			udiTmpDWord := DINT_TO_UDINT(REAL_TO_DINT(Distance * 10000)); (*Distance*)
			Axis.PlcToDrv.MCParaWord0 := UDINT_TO_UINT(udiTmpDWord);
			Axis.PlcToDrv.MCParaWord1 := UDINT_TO_UINT(ROR(udiTmpDWord,16));

			udiTmpDWord := DINT_TO_UDINT(REAL_TO_DINT(Velocity * 1000000)); (*Maximal velocity*)
			Axis.PlcToDrv.MCParaWord2 := UDINT_TO_UINT(udiTmpDWord);
			Axis.PlcToDrv.MCParaWord3 := UDINT_TO_UINT(ROR(udiTmpDWord,16));

			udiTmpDWord := DINT_TO_UDINT(REAL_TO_DINT(Acceleration * 100000)); (*Acceleration*)
			Axis.PlcToDrv.MCParaWord4 := UDINT_TO_UINT(udiTmpDWord);
			Axis.PlcToDrv.MCParaWord5 := UDINT_TO_UINT(ROR(udiTmpDWord,16));

			udiTmpDWord := DINT_TO_UDINT(REAL_TO_DINT(Deceleration * 100000)); (*Deceleration*)
			Axis.PlcToDrv.MCParaWord6 := UDINT_TO_UINT(udiTmpDWord);
			Axis.PlcToDrv.MCParaWord7 := UDINT_TO_UINT(ROR(udiTmpDWord,16));

			udiTmpDWord := DINT_TO_UDINT(REAL_TO_DINT(Jerk * 10000)); (*Jerk*)
			Axis.PlcToDrv.MCParaWord8 := UDINT_TO_UINT(udiTmpDWord);
			Axis.PlcToDrv.MCParaWord9 := UDINT_TO_UINT(ROR(udiTmpDWord,16));
			
			LM_UptMCI(Axis);
			
			uiFbState := 2;
		ELSE
			Axis.CommandRunning := FALSE;
			uiFbState := 50; (*Error state*)
			Error := TRUE;
			ErrorID := 16#06; (*Invalid input(s)*)
		END_IF

	2:	(*Prüfen ob Befehl ausgeführt ][ Check if command has been executed*)
		IF usiOldCmdCount = usiNewCmdCount AND uiCState = 16#08 AND Axis.DrvToPlc.StateVar.6 THEN
			Done := TRUE;
			Busy := FALSE;
			Axis.PlcToDrv.MCHeader := 16#0000 + usiNewCmdCount; (*Send no operation*)
			Axis.CommandRunning := FALSE;
			uiFbState := 3;
		END_IF

	3:	IF NOT Execute THEN
			uiFbState := 0;
			Busy := FALSE;
			Done := FALSE;
		END_IF

	50:	Error := TRUE;
		Busy := FALSE;
		Done := FALSE;
		IF NOT Execute THEN
			uiFbState := 0;
			Error := FALSE;
			ErrorID := 0;
		END_IF

END_CASE

END_FUNCTION_BLOCK

// POUs/LinMot MC Function Blocks/LMmt_StartCTCommand
FUNCTION_BLOCK LMmt_StartCTCommand
VAR_INPUT
	Execute			:BOOL;	(*Execute command*)
	CTEntryID		:UINT;	(*ID of the Command Table to be started*)
END_VAR
VAR_IN_OUT
	Axis			:tstLM_Axis; (*Axis reference*)
END_VAR
VAR_OUTPUT
	Done			:BOOL;	(*Command has been executed*)
	Busy			:BOOL;	(*Command running / FB Busy*)
	Error			:BOOL;	(*Error detected*)
	ErrorID			:UINT;	(*Error ID:
							01h: Axis not ready
 							02h: Axis already has command running
 							03h: Axis has error
 							04h: Command interrupted
 							05h: Command aborted
							06h: Invalid input(s)
							*)
END_VAR
VAR
	usiOldCmdCount 	:USINT;	(*internal -> *)
	usiNewCmdCount	:USINT;	(*internal -> *)
	uiCState		:UINT;	(*internal -> *)
	uiFbState		:UINT;	(*internal -> *)
	rTrig			:LM_R_TRIG;	(*internal -> *)

 	uiCmdHeader 	:UINT := 16#2000;	(*CommandHeader (200xh) of the "Start Command Table Command (200xh)" motion command*)
END_VAR
(*Version history:
Date         	 | Version    		| Created under     	| Author          	| Remark 
------------------------------------------------------------------------------------------------------------------------------- 
2011-jul-12   	 | 1.0.0      		| V2.11.0 (Build 1016)	| fj  				| initial release
2011-sep-13   	 | 1.0.1      		| V2.11.0 (Build 1016)	| fj  				| removed check for "StandStill_LM" on Execute rising edge 
2011-dec-01   	 | 1.0.2      		| V2.11.0 (Build 1016)	| fj  				| code optimisation
2012-apr-25   	 | 1.1.0     		| V2.11.0 (Build 1016)	| fj  				| added input parameters check
*)

(*Variablen ][ variables*)
usiOldCmdCount := SHR(UINT_TO_USINT(SHL(Axis.DrvToPlc.StateVar,4)),4);
uiCState := SHR(Axis.DrvToPlc.StateVar, 8);

(*Flankenerkennung am Execute Eingang*)
(*Edge detection on Execute input*)
rTrig(CLK:=Execute);
IF rTrig.Q AND uiCState = 16#08 AND NOT Axis.CommandRunning THEN (*Start command*)
	Axis.CommandRunning := TRUE;
	Busy := TRUE;
	uiFbState := 1;
ELSIF rTrig.Q AND Busy THEN (*Restart command / New rising edge on execute input*)
	Axis.CommandRunning := TRUE;
	Busy := TRUE;
	uiFbState := 1;
ELSIF rTrig.Q AND uiCState <> 16#08 THEN (*Axis not ready*)
	uiFbState := 50; (*Error state*)
	Error := TRUE;
	ErrorID := 16#01; (*Axis not ready*)
ELSIF rTrig.Q AND Axis.CommandRunning AND NOT Busy THEN (*Axis already has a command running*)
	uiFbState := 50; (*Error state*)
	Error := TRUE;
	ErrorID := 16#02; (*Axis already has a command running*)
END_IF

IF Busy AND uiCState = 16#04 THEN
	Axis.CommandRunning := FALSE;
	uiFbState := 50;
	Error := TRUE;
	ErrorID := 16#03; (*Axis has error*)
END_IF

IF Busy AND uiCState <> 16#08 THEN
	Axis.CommandRunning := FALSE;
	uiFbState := 50; (*Error state*)
	Error := TRUE;
	ErrorID := 16#04; (*Command interupted*)
ELSIF Busy AND Axis.CommandAborted THEN
	uiFbState := 50; (*Error state*)
	Error := TRUE;
	ErrorID := 16#05; (*Command aborted*)
END_IF

(*State machine*)
CASE uiFbState OF
	0:	;

	1:	(*Check inputs on valid value*)
		IF (1 <= CTEntryID AND CTEntryID <= 255)
			THEN
			(*Befehlskopf mit CMD Count berechen und senden ][ Calculate and send command header*)
			usiNewCmdCount := (usiOldCmdCount + 1) MOD 16 ; (*MOD 16*)
			Axis.PlcToDrv.MCHeader := 16#0000; (*Reset Header*)
			Axis.PlcToDrv.MCHeader := uiCmdHeader + usiNewCmdCount;

			Axis.PlcToDrv.MCParaWord0 := CTEntryID; (*CTEntryID (line number)*)

			LM_UptMCI(Axis);

			uiFbState := 2;
		ELSE
			Axis.CommandRunning := FALSE;
			uiFbState := 50; (*Error state*)
			Error := TRUE;
			ErrorID := 16#06; (*Invalid input(s)*)
		END_IF

	2:	(*Prüfen ob Befehl ausgeführt ][ Check if command has been executed*)
		IF usiOldCmdCount = usiNewCmdCount AND uiCState = 16#08 THEN
			Done := TRUE;
			Busy := FALSE;
			Axis.PlcToDrv.MCHeader := 16#0000 + usiNewCmdCount; (*Send no operation*)
			Axis.CommandRunning := FALSE;
			uiFbState := 3;
		END_IF

	3:	IF NOT Execute THEN
			uiFbState := 0;
			Busy := FALSE;
			Done := FALSE;
		END_IF

	50:	Error := TRUE;
		Busy := FALSE;
		Done := FALSE;
		IF NOT Execute THEN
			uiFbState := 0;
			Error := FALSE;
			ErrorID := 0;
		END_IF

END_CASE

END_FUNCTION_BLOCK

// POUs/LinMot MC Function Blocks/LMmt_WriteLivePar
FUNCTION_BLOCK LMmt_WriteLivePar
VAR_INPUT
	Execute			:BOOL;	(*Execute command*)
	UPID			:UINT;	(*Parameter ID (UPID = Unique Parameter ID*)
	UPIDValue		:DINT;	(*Parameter value*)
END_VAR
VAR_IN_OUT
	Axis			:tstLM_Axis; (*Axis reference*)
END_VAR
VAR_OUTPUT
	Done			:BOOL;	(*Command has been executed*)
	Busy			:BOOL;	(*Command running / FB Busy*)
	Error			:BOOL;	(*Error detected*)
	ErrorID			:UINT;	(*Error ID:
							01h: Axis not ready
 							02h: Axis already has command running
 							03h: Axis has error
 							04h: Command interrupted
 							05h: Command aborted
							06h: Invalid input(s)
							*)
END_VAR
VAR
	usiOldCmdCount 	:USINT;	(*internal -> *)
	usiNewCmdCount	:USINT;	(*internal -> *)
	uiCState		:UINT;	(*internal -> *)
	uiFbState		:UINT;	(*internal -> *)
	rTrig			:LM_R_TRIG;	(*internal -> *)
	udiTmpDWord		:UDINT;	(*internal -> *)

 	uiCmdHeader 	:UINT := 16#0020;	(*CommandHeader (002xh) of the "Write Live Parameter (002xh)" motion command*)
END_VAR
(*Version history:
Date         	 | Version    		| Created under     	| Author          	| Remark 
------------------------------------------------------------------------------------------------------------------------------- 
2011-jul-12   	 | 1.0.0      		| V2.11.0 (Build 1016)	| fj  				| initial release 
2011-dec-01   	 | 1.0.2      		| V2.11.0 (Build 1016)	| fj  				| code optimisation
2012-apr-25   	 | 1.1.0     		| V2.11.0 (Build 1016)	| fj  				| added input parameters check
*)

(*Variablen ][ variables*)
usiOldCmdCount := SHR(UINT_TO_USINT(SHL(Axis.DrvToPlc.StateVar,4)),4);
uiCState := SHR(Axis.DrvToPlc.StateVar, 8);

(*Flankenerkennung am Execute Eingang*)
(*Edge detection on Execute input*)
rTrig(CLK:=Execute);
IF rTrig.Q AND uiCState = 16#08 AND NOT Axis.CommandRunning THEN (*Start command*)
	Axis.CommandRunning := TRUE;
	Busy := TRUE;
	uiFbState := 1;
ELSIF rTrig.Q AND Busy THEN (*Restart command / New rising edge on execute input*)
	Axis.CommandRunning := TRUE;
	Busy := TRUE;
	uiFbState := 1;
ELSIF rTrig.Q AND uiCState <> 16#08 THEN (*Axis not ready*)
	uiFbState := 50; (*Error state*)
	Error := TRUE;
	ErrorID := 16#01; (*Axis not ready*)
ELSIF rTrig.Q AND Axis.CommandRunning AND NOT Busy THEN (*Axis already has a command running*)
	uiFbState := 50; (*Error state*)
	Error := TRUE;
	ErrorID := 16#02; (*Axis already has a command running*)
END_IF

IF Busy AND uiCState = 16#04 THEN
	Axis.CommandRunning := FALSE;
	uiFbState := 50;
	Error := TRUE;
	ErrorID := 16#03; (*Axis has error*)
END_IF

IF Busy AND uiCState <> 16#08 THEN
	Axis.CommandRunning := FALSE;
	uiFbState := 50; (*Error state*)
	Error := TRUE;
	ErrorID := 16#04; (*Command interupted*)
ELSIF Busy AND Axis.CommandAborted THEN
	uiFbState := 50; (*Error state*)
	Error := TRUE;
	ErrorID := 16#05; (*Command aborted*)
END_IF

(*State machine*)
CASE uiFbState OF
	0:	;

	1:	(*Check inputs on valid value*)
		IF (0 < UPID AND UPID <= 65535)
			AND (-2147483648 <= UPIDValue AND UPIDValue <= 2147483647)
			THEN
			(*Befehlskopf mit CMD Count berechen und senden ][ Calculate and send command header*)
			usiNewCmdCount  := (usiOldCmdCount + 1) MOD 16 ; (*MOD 16*)
			Axis.PlcToDrv.MCHeader := 16#0000; (*Reset Header*)
			Axis.PlcToDrv.MCHeader := uiCmdHeader + usiNewCmdCount;

			Axis.PlcToDrv.MCParaWord0 := UPID; (*UPID number*)

			udiTmpDWord := DINT_TO_UDINT(UPIDValue); (*UPID parameter value*)
			Axis.PlcToDrv.MCParaWord1 := UDINT_TO_UINT(udiTmpDWord);
			Axis.PlcToDrv.MCParaWord2 := UDINT_TO_UINT(ROR(udiTmpDWord,16));

			LM_UptMCI(Axis);

			uiFbState := 2;
		ELSE
			Axis.CommandRunning := FALSE;
			uiFbState := 50; (*Error state*)
			Error := TRUE;
			ErrorID := 16#06; (*Invalid input(s)*)
		END_IF

	2:	(*Prüfen ob Befehl ausgeführt ][ Check if command has been executed*)
		IF usiOldCmdCount = usiNewCmdCount AND uiCState = 16#08 THEN
			Done := TRUE;
			Busy := FALSE;
			Axis.PlcToDrv.MCHeader := 16#0000 + usiNewCmdCount; (*Send no operation*)
			Axis.CommandRunning := FALSE;
			uiFbState := 3;
		END_IF

	3:	IF NOT Execute THEN
			uiFbState := 0;
			Busy := FALSE;
			Done := FALSE;
		END_IF

	50:	Error := TRUE;
		Busy := FALSE;
		Done := FALSE;
		IF NOT Execute THEN
			uiFbState := 0;
			Error := FALSE;
			ErrorID := 0;
		END_IF

END_CASE

END_FUNCTION_BLOCK

// POUs/LinMot MC Function Blocks Advanced/Unofficial_Unsupported/LMav_PVStreamLREAL
FUNCTION_BLOCK LMav_PVStreamLREAL
VAR_INPUT
	Enable 			:BOOL;	(*Enable PV streaming*)
	Position		:LREAL;	(*Setpoint position in [mm]*)
	Velocity		:LREAL;	(*Setpoint velocity in [mm/s]*)
END_VAR
VAR_IN_OUT
	Axis 			:tstLM_Axis; (*Axis*)
END_VAR
VAR_OUTPUT
	Streaming 		:BOOL;	(*Streaming / FB Busy*)
	Error 			:BOOL;	(*Error detected*)
	ErrorID			:UINT;	(*Error ID:
							01h: Axis not ready
 							02h: Axis already has command running
 							03h: Axis has error
 							04h: Command interrupted
 							05h: Command aborted
							06h: Invalid input(s)
							*)
END_VAR
VAR
	uiCState		:UINT;	(*internal -> *)
	uiFbState 		:UINT;	(*internal -> *)
	rTrig 			:LM_R_TRIG;	(*internal -> *)
	udiTmpDWord		:UDINT;	(*internal -> *)
	bTemp			:BOOL;	(*internal -> *)

	uiCmdHeader 	:UINT := 16#0310; (*internal -> CommandHeader (031xh) of the "PV Stream With Slave Generated Time Stamp (031xh)" motion command*)
END_VAR
(*Version history:
Date         	 | Version    		| Created under     	| Author          	| Remark 
------------------------------------------------------------------------------------------------------------------------------- 
2011-jul-20   	 | 1.0.0      		| V2.11.0 (Build 1016)	| fj  				| initial release
2011-sep-13   	 | 1.0.1      		| V2.11.0 (Build 1016)	| fj  				| removed check for "StandStill_LM" on Enable rising edge
2011-dec-01   	 | 1.0.2      		| V2.11.0 (Build 1016)	| fj  				| code optimisation
2012-apr-25   	 | 1.1.0     		| V2.11.0 (Build 1016)	| fj  				| removed input range check (position&velocity) / changed input data types REAL to LREAL
*)

(*Variablen ][ variables*)
uiCState := SHR(Axis.DrvToPlc.StateVar, 8);

(*Flankenerkennung am Execute Eingang*)
(*Edge detection on Execute input*)
rTrig(CLK:=Enable);
IF rTrig.Q AND uiCState = 16#08 AND NOT Axis.CommandRunning THEN (*Start command*)
	Axis.CommandRunning := TRUE;
	uiFbState := 1;
ELSIF rTrig.Q AND uiCState <> 16#08 THEN (*Axis not ready*)
	uiFbState := 50; (*Error state*)
	Error := TRUE;
	ErrorID := 16#01; (*Axis not ready*)
ELSIF rTrig.Q AND Axis.CommandRunning THEN (*Axis already has a command running*)
	uiFbState := 50; (*Error state*)
	Error := TRUE;
	ErrorID := 16#02; (*Axis already has a command running*)
END_IF

IF Streaming AND uiCState = 16#04 THEN
	Axis.CommandRunning := FALSE;
	uiFbState := 50;
	Error := TRUE;
	ErrorID := 16#03; (*Axis has error*)
END_IF

IF Streaming AND uiCState <> 16#08 THEN
	Axis.CommandRunning := FALSE;
	uiFbState := 50; (*Error state*)
	Error := TRUE;
	ErrorID := 16#04; (*Command interupted*)
ELSIF Streaming AND Axis.CommandAborted THEN
	uiFbState := 50; (*Error state*)
	Error := TRUE;
	ErrorID := 16#05; (*Command aborted*)
END_IF

(*uiState machine*)
CASE uiFbState OF
	0:	;

	1:	(*Check inputs on valid value*)
		(*Streaming*)
		bTemp := Axis.PlcToDrv.MCHeader.0;
		Axis.PlcToDrv.MCHeader := uiCmdHeader;
		Axis.PlcToDrv.MCHeader.0 := NOT bTemp;

		(*Parameter Umrechung*)
		(*Calculate parameters*)
		udiTmpDWord := DINT_TO_UDINT(LREAL_TO_DINT(Position * 10000)); (*Position*)
		Axis.PlcToDrv.MCParaWord0 := UDINT_TO_UINT(udiTmpDWord);
		Axis.PlcToDrv.MCParaWord1 := UDINT_TO_UINT(ROR(udiTmpDWord,16));

		udiTmpDWord := DINT_TO_UDINT(LREAL_TO_DINT(Velocity * 1000)); (*Velocity*)
		Axis.PlcToDrv.MCParaWord2 := UDINT_TO_UINT(udiTmpDWord);
		Axis.PlcToDrv.MCParaWord3 := UDINT_TO_UINT(ROR(udiTmpDWord,16));

		LM_UptMCI(Axis);

		Streaming := TRUE;
	
		IF NOT Enable THEN
			uiFbState := 2;
		END_IF

	2:	(*Stop streaming*)
		bTemp := Axis.PlcToDrv.MCHeader.0;
		Axis.PlcToDrv.MCHeader := 16#03F0; (*Header 03F0h (Stop Stream)*)
		Axis.PlcToDrv.MCHeader.0 := NOT bTemp;

		uiFbState := 3;

	3:	IF Axis.PlcToDrv.MCHeader.0 = Axis.DrvToPlc.StateVar.0 THEN
			Streaming := FALSE;
			Axis.PlcToDrv.MCHeader := 16#0000; (*No Operation*)
			Axis.PlcToDrv.MCHeader.0 := Axis.DrvToPlc.StateVar.0;
			Axis.CommandRunning := FALSE;
			uiFbState := 0;
		END_IF

	50:	Error := TRUE;
		Axis.PlcToDrv.MCHeader := 16#0000; (*No Operation*)
		Streaming := FALSE;
		uiFbState := 51;

	51:	 IF NOT Enable THEN
			uiFbState := 0;
			Error := FALSE;
			ErrorID := 0;
		END_IF

END_CASE

END_FUNCTION_BLOCK

// POUs/LinMot MC Function Blocks Advanced/LMav_CurrentCmdMode
FUNCTION_BLOCK LMav_CurrentCmdMode
VAR_INPUT
	Enable 			:BOOL;	(*Enable current streaming*)
	Current			:REAL;	(*Setpoint Current*)
END_VAR
VAR_IN_OUT
	Axis 			:tstLM_Axis; (*Axis reference*)
END_VAR
VAR_OUTPUT
	Streaming 		:BOOL;	(*Streaming / FB Busy*)
	Error 			:BOOL;	(*Error detected*)
	ErrorID			:UINT;	(*Error ID:
							01h: Axis not ready
 							02h: Axis already has command running
 							03h: Axis has error
 							04h: Command interrupted
 							05h: Command aborted
							06h: Invalid input(s)
							*)
END_VAR
VAR
	uiCState		:UINT;	(*internal -> *)
	uiFbState 		:UINT;	(*internal -> *)
	rTrig 			:LM_R_TRIG;	(*internal -> *)
	udiTmpDWord		:UDINT;	(*internal -> *)
	bTemp			:BOOL;	(*internal -> *)

	uiCmdHeader 	:UINT := 16#3900; (*internal -> CommandHeader (390xh) of the "Current Command Mode (390xh)" motion command*)
END_VAR
(*Version history:
Date         	 | Version    		| Created under     	| Author          	| Remark 
------------------------------------------------------------------------------------------------------------------------------- 
2011-jul-20   	 | 1.0.0      		| V2.11.0 (Build 1016)	| fj  				| initial release
2011-sep-13   	 | 1.0.1      		| V2.11.0 (Build 1016)	| fj  				| removed check for "StandStill_LM" on Execute rising edge
2011-dec-01   	 | 1.0.2      		| V2.11.0 (Build 1016)	| fj  				| code optimisation
2012-apr-25   	 | 1.1.0     		| V2.11.0 (Build 1016)	| fj  				| added input parameters check
*)

(*Variablen ][ variables*)
uiCState := SHR(Axis.DrvToPlc.StateVar, 8);

(*Flankenerkennung am Execute Eingang*)
(*Edge detection on Execute input*)
rTrig(CLK:=Enable);
IF rTrig.Q AND uiCState = 16#08 AND NOT Axis.CommandRunning THEN (*Start command*)
	Axis.CommandRunning := TRUE;
	uiFbState := 1;
ELSIF rTrig.Q AND uiCState <> 16#08 THEN (*Axis not ready*)
	uiFbState := 50; (*Error state*)
	Error := TRUE;
	ErrorID := 16#01; (*Axis not ready*)
ELSIF rTrig.Q AND Axis.CommandRunning THEN (*Axis already has a command running*)
	uiFbState := 50; (*Error state*)
	Error := TRUE;
	ErrorID := 16#02; (*Axis already has a command running*)
END_IF

IF Streaming AND uiCState = 16#04 THEN
	Axis.CommandRunning := FALSE;
	uiFbState := 50;
	Error := TRUE;
	ErrorID := 16#03; (*Axis has error*)
END_IF

IF Streaming AND uiCState <> 16#08 THEN
	Axis.CommandRunning := FALSE;
	uiFbState := 50; (*Error state*)
	Error := TRUE;
	ErrorID := 16#04; (*Command interupted*)
ELSIF Streaming AND Axis.CommandAborted THEN
	uiFbState := 50; (*Error state*)
	Error := TRUE;
	ErrorID := 16#05; (*Command aborted*)
END_IF

(*uiState machine*)
CASE uiFbState OF
	0:	;

	1:	(*Check inputs on valid value*)
		IF (-2147483.0 <= Current AND Current <= 2147483.0)
			THEN
			(*Streaming*)
			bTemp := Axis.PlcToDrv.MCHeader.0;
			Axis.PlcToDrv.MCHeader := uiCmdHeader;
			Axis.PlcToDrv.MCHeader.0 := NOT bTemp;

			(*Parameter Umrechung*)
			(*Calculate parameters*)
			udiTmpDWord := DINT_TO_UDINT(REAL_TO_DINT(Current * 1000)); (*Current*)
			Axis.PlcToDrv.MCParaWord0 := UDINT_TO_UINT(udiTmpDWord);
			Axis.PlcToDrv.MCParaWord1 := UDINT_TO_UINT(ROR(udiTmpDWord,16));

			LM_UptMCI(Axis);

			Streaming := TRUE;

			IF NOT Enable THEN
				uiFbState := 2;
			END_IF
		ELSE
			Axis.CommandRunning := FALSE;
			uiFbState := 50; (*Error state*)
			Error := TRUE;
			ErrorID := 16#06; (*Invalid input(s)*)
		END_IF

	2:	(*Stop streaming*)
		bTemp := Axis.PlcToDrv.MCHeader.0;
		Axis.PlcToDrv.MCHeader := 16#39F0; (*Header 39Fxh (Change to Position Controlled mode)*)
		Axis.PlcToDrv.MCHeader.0 := NOT bTemp;

		uiFbState := 3;

	3:	IF Axis.PlcToDrv.MCHeader.0 = Axis.DrvToPlc.StateVar.0 THEN
			Streaming := FALSE;
			Axis.CommandRunning := FALSE;
			Axis.PlcToDrv.MCHeader := 16#0000; (*No Operation*)
			Axis.PlcToDrv.MCHeader.0 := Axis.DrvToPlc.StateVar.0;
			uiFbState := 0;
		END_IF

	50:	Error := TRUE;
		Axis.PlcToDrv.MCHeader := 16#0000; (*No Operation*)
		Streaming := FALSE;
		uiFbState := 51;

	51:	 IF NOT Enable THEN
			uiFbState := 0;
			Error := FALSE;
			ErrorID := 0;
		END_IF

END_CASE

END_FUNCTION_BLOCK

// POUs/LinMot MC Function Blocks Advanced/LMav_Mod16BitCTPar
FUNCTION_BLOCK LMav_Mod16BitCTPar
VAR_INPUT
	Execute			:BOOL;	(*Execute command*)
	CTEntryID		:UINT;	(*Line number of the Command Table to be modified*)
	ParaOffset		:UINT;	(*Parameter offset (6 for the first)*)
	ParaValue		:INT;	(*Parameter value*)
END_VAR
VAR_IN_OUT
	Axis			:tstLM_Axis; (*Axis reference*)
END_VAR
VAR_OUTPUT
	Done			:BOOL;	(*Command has been executed*)
	Busy			:BOOL;	(*Command running / FB Busy*)
	Error			:BOOL;	(*Error detected*)
	ErrorID			:UINT;	(*Error ID:
							01h: Axis not ready
 							02h: Axis already has command running
 							03h: Axis has error
 							04h: Command interrupted
 							05h: Command aborted
							06h: Invalid input(s)
							*)
END_VAR
VAR
	usiOldCmdCount 	:USINT;	(*internal -> *)
	usiNewCmdCount	:USINT;	(*internal -> *)
	uiCState		:UINT;	(*internal -> *)
	uiFbState		:UINT;	(*internal -> *)
	rTrig			:LM_R_TRIG;	(*internal -> *)

 	uiCmdHeader 	:UINT := 16#2080;	(*CommandHeader (208xh) of the "Modify Command Table 16 bit Parameter in RAM (208xh)" motion command*)
END_VAR
(*Version history:
Date         	 | Version    		| Created under     	| Author          	| Remark 
------------------------------------------------------------------------------------------------------------------------------- 
2011-jul-12   	 | 1.0.0      		| V2.11.0 (Build 1016)	| fj  				| initial release 
2011-dec-01   	 | 1.0.2      		| V2.11.0 (Build 1016)	| fj  				| code optimisation
2012-apr-25   	 | 1.1.0     		| V2.11.0 (Build 1016)	| fj  				| added input parameters check
*)

(*Variablen ][ variables*)
usiOldCmdCount := SHR(UINT_TO_USINT(SHL(Axis.DrvToPlc.StateVar,4)),4);
uiCState := SHR(Axis.DrvToPlc.StateVar, 8);

(*Flankenerkennung am Execute Eingang*)
(*Edge detection on Execute input*)
rTrig(CLK:=Execute);
IF rTrig.Q AND uiCState = 16#08 AND NOT Axis.CommandRunning THEN (*Start command*)
	Axis.CommandRunning := TRUE;
	Busy := TRUE;
	uiFbState := 1;
ELSIF rTrig.Q AND Busy THEN (*Restart command / New rising edge on execute input*)
	Axis.CommandRunning := TRUE;
	Busy := TRUE;
	uiFbState := 1;
ELSIF rTrig.Q AND uiCState <> 16#08 THEN (*Axis not ready*)
	uiFbState := 50; (*Error state*)
	Error := TRUE;
	ErrorID := 16#01; (*Axis not ready*)
ELSIF rTrig.Q AND Axis.CommandRunning AND NOT Busy THEN (*Axis already has a command running*)
	uiFbState := 50; (*Error state*)
	Error := TRUE;
	ErrorID := 16#02; (*Axis already has a command running*)
END_IF

IF Busy AND uiCState = 16#04 THEN
	Axis.CommandRunning := FALSE;
	uiFbState := 50;
	Error := TRUE;
	ErrorID := 16#03; (*Axis has error*)
END_IF

IF Busy AND uiCState <> 16#08 THEN
	Axis.CommandRunning := FALSE;
	uiFbState := 50; (*Error state*)
	Error := TRUE;
	ErrorID := 16#04; (*Command interupted*)
ELSIF Busy AND Axis.CommandAborted THEN
	uiFbState := 50; (*Error state*)
	Error := TRUE;
	ErrorID := 16#05; (*Command aborted*)
END_IF

(*State machine*)
CASE uiFbState OF
	0:	;

	1:	(*Check inputs on valid value*)
		IF (0 < CTEntryID AND CTEntryID <= 255)
			AND (0 <= ParaOffset AND ParaOffset <= 20)
			AND (-32768 <= ParaValue AND ParaValue <= 32767)
			THEN
			(*Befehlskopf mit CMD Count berechen und senden ][ Calculate and send command header*)
			usiNewCmdCount := (usiOldCmdCount + 1) MOD 16; (*MOD 16*)
			Axis.PlcToDrv.MCHeader := 16#0000; (*Reset Header*)
			Axis.PlcToDrv.MCHeader := uiCmdHeader + usiNewCmdCount;

			Axis.PlcToDrv.MCParaWord0 := CTEntryID; (*CT_EntryID*)
			Axis.PlcToDrv.MCParaWord1 := ParaOffset; (*Parameter offset*)
			Axis.PlcToDrv.MCParaWord2 := INT_TO_UINT(ParaValue); (*Parameter value*)

			LM_UptMCI(Axis);

			uiFbState := 2;
		ELSE
			Axis.CommandRunning := FALSE;
			uiFbState := 50; (*Error state*)
			Error := TRUE;
			ErrorID := 16#06; (*Invalid input(s)*)
		END_IF

	2:	(*Prüfen ob Befehl ausgeführt ][ Check if command has been executed*)
		IF usiOldCmdCount = usiNewCmdCount AND uiCState = 16#08 THEN
			Done := TRUE;
			Busy := FALSE;
			Axis.PlcToDrv.MCHeader := 16#0000 + usiNewCmdCount; (*Send no operation*)
			Axis.CommandRunning := FALSE;
			uiFbState := 3;
		END_IF

	3:	IF NOT Execute THEN
			uiFbState := 0;
			Busy := FALSE;
			Done := FALSE;
		END_IF

	50:	Error := TRUE;
		Busy := FALSE;
		Done := FALSE;
		IF NOT Execute THEN
			uiFbState := 0;
			Error := FALSE;
			ErrorID := 0;
		END_IF

END_CASE

END_FUNCTION_BLOCK

// POUs/LinMot MC Function Blocks Advanced/LMav_Mod32BitCTPar
FUNCTION_BLOCK LMav_Mod32BitCTPar
VAR_INPUT
	Execute			:BOOL;	(*Execute command*)
	CTEntryID		:UINT;	(*Line number of the Command Table to be modified*)
	ParaOffset		:UINT;	(*Parameter offset (6 for the first)*)
	ParaValue		:DINT;	(*Parameter value*)
END_VAR
VAR_IN_OUT
	Axis			:tstLM_Axis; (*Axis reference*)
END_VAR
VAR_OUTPUT
	Done			:BOOL;	(*Command has been executed*)
	Busy			:BOOL;	(*Command running / FB Busy*)
	Error			:BOOL;	(*Error detected*)
	ErrorID			:UINT;	(*Error ID:
							01h: Axis not ready
 							02h: Axis already has command running
 							03h: Axis has error
 							04h: Command interrupted
 							05h: Command aborted
							06h: Invalid input(s)
							*)
END_VAR
VAR
	usiOldCmdCount 	:USINT;	(*internal -> *)
	usiNewCmdCount	:USINT;	(*internal -> *)
	uiCState		:UINT;	(*internal -> *)
	uiFbState		:UINT;	(*internal -> *)
	rTrig			:LM_R_TRIG;	(*internal -> *)
	udiTmpDWord		:UDINT;	(*internal -> *)

 	uiCmdHeader 	:UINT := 16#2090; 	(*CommandHeader (209xh) of the "Modify Command Table 32 bit Parameter in RAM (209xh)" motion command*)
END_VAR
(*Version history:
Date         	 | Version    		| Created under     	| Author          	| Remark 
------------------------------------------------------------------------------------------------------------------------------- 
2011-jul-12   	 | 1.0.0      		| V2.11.0 (Build 1016)	| fj  				| initial release 
2011-dec-01   	 | 1.0.2      		| V2.11.0 (Build 1016)	| fj  				| code optimisation
2012-apr-25   	 | 1.1.0     		| V2.11.0 (Build 1016)	| fj  				| added input parameters check
*)

(*Variablen ][ variables*)
usiOldCmdCount := SHR(UINT_TO_USINT(SHL(Axis.DrvToPlc.StateVar,4)),4);
uiCState := SHR(Axis.DrvToPlc.StateVar, 8);

(*Flankenerkennung am Execute Eingang*)
(*Edge detection on Execute input*)
rTrig(CLK:=Execute);
IF rTrig.Q AND uiCState = 16#08 AND NOT Axis.CommandRunning THEN (*Start command*)
	Axis.CommandRunning := TRUE;
	Busy := TRUE;
	uiFbState := 1;
ELSIF rTrig.Q AND Busy THEN (*Restart command / New rising edge on execute input*)
	Axis.CommandRunning := TRUE;
	Busy := TRUE;
	uiFbState := 1;
ELSIF rTrig.Q AND uiCState <> 16#08 THEN (*Axis not ready*)
	uiFbState := 50; (*Error state*)
	Error := TRUE;
	ErrorID := 16#01; (*Axis not ready*)
ELSIF rTrig.Q AND Axis.CommandRunning AND NOT Busy THEN (*Axis already has a command running*)
	uiFbState := 50; (*Error state*)
	Error := TRUE;
	ErrorID := 16#02; (*Axis already has a command running*)
END_IF

IF Busy AND uiCState = 16#04 THEN
	Axis.CommandRunning := FALSE;
	uiFbState := 50;
	Error := TRUE;
	ErrorID := 16#03; (*Axis has error*)
END_IF

IF Busy AND uiCState <> 16#08 THEN
	Axis.CommandRunning := FALSE;
	uiFbState := 50; (*Error state*)
	Error := TRUE;
	ErrorID := 16#04; (*Command interupted*)
ELSIF Busy AND Axis.CommandAborted THEN
	uiFbState := 50; (*Error state*)
	Error := TRUE;
	ErrorID := 16#05; (*Command aborted*)
END_IF

(*State machine*)
CASE uiFbState OF
	0:	;

	1:	(*Check inputs on valid value*)
		IF (0 < CTEntryID AND CTEntryID <= 255)
			AND (0 <= ParaOffset AND ParaOffset <= 20)
			AND (-2147483648 <= ParaValue AND ParaValue <= 2147483647)
			THEN
			(*Befehlskopf mit CMD Count berechen und senden ][ Calculate and send command header*)
			usiNewCmdCount := (usiOldCmdCount + 1) MOD 16 ; (*MOD 16*)
			Axis.PlcToDrv.MCHeader := 16#0000; (*Reset Header*)
			Axis.PlcToDrv.MCHeader := uiCmdHeader + usiNewCmdCount;

			Axis.PlcToDrv.MCParaWord0 := CTEntryID; (*CT_EntryID*)
			Axis.PlcToDrv.MCParaWord1 := ParaOffset; (*Parameter offset*)

			udiTmpDWord := DINT_TO_UDINT(ParaValue);(*Parameter value*)
			Axis.PlcToDrv.MCParaWord2 := UDINT_TO_UINT(udiTmpDWord);
			Axis.PlcToDrv.MCParaWord3 := UDINT_TO_UINT(ROR(udiTmpDWord,16));

			LM_UptMCI(Axis);

			uiFbState := 2;
		ELSE
			Axis.CommandRunning := FALSE;
			uiFbState := 50; (*Error state*)
			Error := TRUE;
			ErrorID := 16#06; (*Invalid input(s)*)
		END_IF

	2:	(*Prüfen ob Befehl ausgeführt ][ Check if command has been executed*)
		IF usiOldCmdCount = usiNewCmdCount AND uiCState = 16#08 THEN
			Done := TRUE;
			Busy := FALSE;
			Axis.PlcToDrv.MCHeader := 16#0000 + usiNewCmdCount; (*Send no operation*)
			Axis.CommandRunning := FALSE;
			uiFbState := 3;
		END_IF

	3:	IF NOT Execute THEN
			uiFbState := 0;
			Busy := FALSE;
			Done := FALSE;
		END_IF

	50:	Error := TRUE;
		Busy := FALSE;
		Done := FALSE;
		IF NOT Execute THEN
			uiFbState := 0;
			Error := FALSE;
			ErrorID := 0;
		END_IF

END_CASE

END_FUNCTION_BLOCK

// POUs/LinMot MC Function Blocks Advanced/LMav_MoveBestehorn
FUNCTION_BLOCK LMav_MoveBestehorn
VAR_INPUT
	Execute			:BOOL;	(*Execute command*)
	Position		:REAL;	(*Target position in [mm]*)
	Velocity		:REAL;	(*Maximal velocity in [m/s]*)
	Acceleration	:REAL;	(*Acceleration in [m/s^2]*)
	Jerk			:REAL;	(*Maximal jerk in [m/s^3]*)
END_VAR
VAR_IN_OUT
	Axis			:tstLM_Axis; (*Axis reference*)
END_VAR
VAR_OUTPUT
	Done			:BOOL;	(*Command has been executed*)
	Busy			:BOOL;	(*Command running / FB Busy*)
	Error           		:BOOL;	(*Error detected*)
	ErrorID 			:UINT;	(*Error ID:
							01h: Axis not ready
 							02h: Axis already has command running
 							03h: Axis has error
 							04h: Command interrupted
 							05h: Command aborted
							06h: Invalid input(s)
							*)
END_VAR
VAR
	usiOldCmdCount 	:USINT;	(*internal -> *)
	usiNewCmdCount	:USINT; 	(*internal -> *)
	uiCState           		:UINT;     	(*internal -> *)
	uiFbState		:UINT;	(*internal -> *)
	rTrig     	    		:LM_R_TRIG;	(*internal -> *)
	udiTmpDWord	:UDINT;	(*internal -> *)

 	uiCmdHeader 	:UINT := 16#0F00;	(*CommandHeader (0F0xh) of the "Bestehorn VAJ Go To Pos (0F0xh)" motion command*)
END_VAR
(*Version history:
Date         	 | Version    		| Created under     	| Author          	| Remark 
------------------------------------------------------------------------------------------------------------------------------- 
2011-jul-12   	 | 1.0.0      		| V2.11.0 (Build 1016)	| fj  				| initial release 
2011-sep-13   	 | 1.0.1      		| V2.11.0 (Build 1016)	| fj  				| removed check for "StandStill_LM" on Execute rising edge
2011-dec-01   	 | 1.0.2      		| V2.11.0 (Build 1016)	| fj  				| code optimisation
2012-apr-25   	 | 1.1.0     		| V2.11.0 (Build 1016)	| fj  				| added input parameters check
*)

(*Variablen ][ variables*)
usiOldCmdCount := SHR(UINT_TO_USINT(SHL(Axis.DrvToPlc.StateVar,4)),4);
uiCState := SHR(Axis.DrvToPlc.StateVar, 8);

(*Flankenerkennung am Execute Eingang*)
(*Edge detection on Execute input*)
rTrig(CLK:=Execute);
IF rTrig.Q AND uiCState = 16#08 AND NOT Axis.CommandRunning THEN (*Start command*)
	Axis.CommandRunning := TRUE;
	Busy := TRUE;
	uiFbState := 1;
ELSIF rTrig.Q AND Busy THEN (*Restart command / New rising edge on execute input*)
	Axis.CommandRunning := TRUE;
	Busy := TRUE;
	uiFbState := 1;
ELSIF rTrig.Q AND uiCState <> 16#08 THEN (*Axis not ready*)
	uiFbState := 50; (*Error state*)
	Error := TRUE;
	ErrorID := 16#01; (*Axis not ready*)
ELSIF rTrig.Q AND Axis.CommandRunning AND NOT Busy THEN (*Axis already has a command running*)
	uiFbState := 50; (*Error state*)
	Error := TRUE;
	ErrorID := 16#02; (*Axis already has a command running*)
END_IF

IF Busy AND uiCState = 16#04 THEN
	Axis.CommandRunning := FALSE;
	uiFbState := 50;
	Error := TRUE;
	ErrorID := 16#03; (*Axis has error*)
END_IF

IF Busy AND uiCState <> 16#08 THEN
	Axis.CommandRunning := FALSE;
	uiFbState := 50; (*Error state*)
	Error := TRUE;
	ErrorID := 16#04; (*Command interupted*)
ELSIF Busy AND Axis.CommandAborted THEN
	uiFbState := 50; (*Error state*)
	Error := TRUE;
	ErrorID := 16#05; (*Command aborted*)
END_IF

(*State machine*)
CASE uiFbState OF
	0:	;

	1:	(*Check inputs on valid value*)
		IF (-214748.0 <= Position AND Position <= 214748.0)
			AND (0.0 < Velocity AND Velocity <= 2147.0)
			AND (0.0 < Acceleration AND Acceleration <= 21474.0)
			AND (0.0 < Jerk AND Jerk <= 214740.0)
			THEN
			(*Befehlskopf mit CMD Count berechen und senden ][ Calculate and send command header*)
			usiNewCmdCount := (usiOldCmdCount + 1) MOD 16 ; (*MOD 16*)
			Axis.PlcToDrv.MCHeader := 16#0000; (*Reset Header*)
			Axis.PlcToDrv.MCHeader := uiCmdHeader + usiNewCmdCount ;

			udiTmpDWord := DINT_TO_UDINT(REAL_TO_DINT(Position * 10000)); (*Target position*)
			Axis.PlcToDrv.MCParaWord0 := UDINT_TO_UINT(udiTmpDWord);
			Axis.PlcToDrv.MCParaWord1 := UDINT_TO_UINT(ROR(udiTmpDWord,16));

			udiTmpDWord := DINT_TO_UDINT(REAL_TO_DINT(Velocity * 1000000)); (*Maximal velocity*)
			Axis.PlcToDrv.MCParaWord2 := UDINT_TO_UINT(udiTmpDWord);
			Axis.PlcToDrv.MCParaWord3 := UDINT_TO_UINT(ROR(udiTmpDWord,16));

			udiTmpDWord := DINT_TO_UDINT(REAL_TO_DINT(Acceleration * 100000)); (*Acceleration*)
			Axis.PlcToDrv.MCParaWord4 := UDINT_TO_UINT(udiTmpDWord);
			Axis.PlcToDrv.MCParaWord5 := UDINT_TO_UINT(ROR(udiTmpDWord,16));

			udiTmpDWord := DINT_TO_UDINT(REAL_TO_DINT(Jerk * 10000)); (*Jerk*)
			Axis.PlcToDrv.MCParaWord6 := UDINT_TO_UINT(udiTmpDWord);
			Axis.PlcToDrv.MCParaWord7 := UDINT_TO_UINT(ROR(udiTmpDWord,16));

			LM_UptMCI(Axis);

			uiFbState := 2;
		ELSE
			Axis.CommandRunning := FALSE;
			uiFbState := 50; (*Error state*)
			Error := TRUE;
			ErrorID := 16#06; (*Invalid input(s)*)
		END_IF

	2:	(*Prüfen ob Befehl ausgeführt ][ Check if command has been executed*)
		IF usiOldCmdCount = usiNewCmdCount AND uiCState = 16#08 AND Axis.DrvToPlc.StateVar.6 THEN
			Done := TRUE;
			Busy := FALSE;
			Axis.PlcToDrv.MCHeader := 16#0000 + usiNewCmdCount; (*Send no operation*)
			Axis.CommandRunning := FALSE;
			uiFbState := 3;
		END_IF

	3:	IF NOT Execute THEN
			uiFbState := 0;
			Busy := FALSE;
			Done := FALSE;
		END_IF

	50:	Error := TRUE;
		Busy := FALSE;
		Done := FALSE;
		IF NOT Execute THEN
			uiFbState := 0;
			Error := FALSE;
			ErrorID := 0;
		END_IF

END_CASE

END_FUNCTION_BLOCK

// POUs/LinMot MC Function Blocks Advanced/LMav_MoveSin
FUNCTION_BLOCK LMav_MoveSin
VAR_INPUT
	Execute			:BOOL;	(*Execute command*)
	Position		:REAL;	(*Target position in [mm]*)
	Velocity		:REAL;	(*Maximal velocity in [m/s]*)
	Acceleration	:REAL;	(*Acceleration in [m/s^2]*)
END_VAR
VAR_IN_OUT
	Axis			:tstLM_Axis; (*Axis reference*)
END_VAR
VAR_OUTPUT
	Done			:BOOL;	(*Command has been executed*)
	Busy			:BOOL;	(*Command running / FB Busy*)
	Error			:BOOL;	(*Error detected*)
	ErrorID			:UINT;	(*Error ID:
							01h: Axis not ready
 							02h: Axis already has command running
 							03h: Axis has error
 							04h: Command interrupted
 							05h: Command aborted
							06h: Invalid input(s)
							*)
END_VAR
VAR
	usiOldCmdCount 	:USINT;	(*internal -> *)
	usiNewCmdCount	:USINT;	(*internal -> *)
	uiCState		:UINT;	(*internal -> *)
	uiFbState		:UINT;	(*internal -> *)
	rTrig			:LM_R_TRIG;	(*internal -> *)
	udiTmpDWord		:UDINT;	(*internal -> *)

 	uiCmdHeader 	:UINT := 16#0E00;	(*CommandHeader (0E0xh) of the "Sin VA Go To Pos (0E0xh)" motion command*)
END_VAR
(*Version history:
Date         	 | Version    		| Created under     	| Author          	| Remark 
------------------------------------------------------------------------------------------------------------------------------- 
2011-jul-12   	 | 1.0.0      		| V2.11.0 (Build 1016)	| fj  				| initial release  
2011-sep-13   	 | 1.0.1      		| V2.11.0 (Build 1016)	| fj  				| removed check for "StandStill_LM" on Execute rising edge
2011-dec-01   	 | 1.0.2      		| V2.11.0 (Build 1016)	| fj  				| code optimisation
2012-apr-25   	 | 1.1.0     		| V2.11.0 (Build 1016)	| fj  				| added input parameters check
*)

(*Variablen ][ variables*)
usiOldCmdCount := SHR(UINT_TO_USINT(SHL(Axis.DrvToPlc.StateVar,4)),4);
uiCState := SHR(Axis.DrvToPlc.StateVar, 8);

(*Flankenerkennung am Execute Eingang*)
(*Edge detection on Execute input*)
rTrig(CLK:=Execute);
IF rTrig.Q AND uiCState = 16#08 AND NOT Axis.CommandRunning THEN (*Start command*)
	Axis.CommandRunning := TRUE;
	Busy := TRUE;
	uiFbState := 1;
ELSIF rTrig.Q AND Busy THEN (*Restart command / New rising edge on execute input*)
	Axis.CommandRunning := TRUE;
	Busy := TRUE;
	uiFbState := 1;
ELSIF rTrig.Q AND uiCState <> 16#08 THEN (*Axis not ready*)
	uiFbState := 50; (*Error state*)
	Error := TRUE;
	ErrorID := 16#01; (*Axis not ready*)
ELSIF rTrig.Q AND Axis.CommandRunning AND NOT Busy THEN (*Axis already has a command running*)
	uiFbState := 50; (*Error state*)
	Error := TRUE;
	ErrorID := 16#02; (*Axis already has a command running*)
END_IF

IF Busy AND uiCState = 16#04 THEN
	Axis.CommandRunning := FALSE;
	uiFbState := 50;
	Error := TRUE;
	ErrorID := 16#03; (*Axis has error*)
END_IF

IF Busy AND uiCState <> 16#08 THEN
	Axis.CommandRunning := FALSE;
	uiFbState := 50; (*Error state*)
	Error := TRUE;
	ErrorID := 16#04; (*Command interupted*)
ELSIF Busy AND Axis.CommandAborted THEN
	uiFbState := 50; (*Error state*)
	Error := TRUE;
	ErrorID := 16#05; (*Command aborted*)
END_IF

(*State machine*)
CASE uiFbState OF
0:	;

1:	(*Check inputs on valid value*)
	IF (-214748.0 <= Position AND Position <= 214748.0)
		AND (0.0 < Velocity AND Velocity <= 2147.0)
		AND (0.0 < Acceleration AND Acceleration <= 21474.0)
		THEN
		(*Befehlskopf mit CMD Count berechen und senden ][ Calculate and send command header*)
		usiNewCmdCount := (usiOldCmdCount + 1) MOD 16 ; (*MOD 16*)
		Axis.PlcToDrv.MCHeader := 16#0000; (*Reset Header*)
		Axis.PlcToDrv.MCHeader := uiCmdHeader + usiNewCmdCount;

		udiTmpDWord := DINT_TO_UDINT(REAL_TO_DINT(Position * 10000)); (*Target position*)
		Axis.PlcToDrv.MCParaWord0 := UDINT_TO_UINT(udiTmpDWord);
		Axis.PlcToDrv.MCParaWord1:= UDINT_TO_UINT(ROR(udiTmpDWord,16));

		udiTmpDWord := DINT_TO_UDINT(REAL_TO_DINT(Velocity * 1000000)); (*Maximal velocity*)
		Axis.PlcToDrv.MCParaWord2 := UDINT_TO_UINT(udiTmpDWord);
		Axis.PlcToDrv.MCParaWord3 := UDINT_TO_UINT(ROR(udiTmpDWord,16));

		udiTmpDWord := DINT_TO_UDINT(REAL_TO_DINT(Acceleration * 100000)); (*Acceleration*)
		Axis.PlcToDrv.MCParaWord4 := UDINT_TO_UINT(udiTmpDWord);
		Axis.PlcToDrv.MCParaWord5 := UDINT_TO_UINT(ROR(udiTmpDWord,16));

		LM_UptMCI(Axis);

		uiFbState := 2;
	ELSE
		Axis.CommandRunning := FALSE;
		uiFbState := 50; (*Error state*)
		Error := TRUE;
		ErrorID := 16#06; (*Invalid input(s)*)
	END_IF

2:	(*Prüfen ob Befehl ausgeführt ][ Check if command has been executed*)
	IF usiOldCmdCount = usiNewCmdCount AND uiCState = 16#08 AND Axis.DrvToPlc.StateVar.6 THEN
		Done := TRUE;
		Busy := FALSE;
		Axis.PlcToDrv.MCHeader := 16#0000 + usiNewCmdCount; (*Send no operation*)
		Axis.CommandRunning := FALSE;
		uiFbState := 3;
	END_IF

3:	IF NOT Execute THEN
		uiFbState := 0;
		Busy := FALSE;
		Done := FALSE;
	END_IF

50:	Error := TRUE;
	Busy := FALSE;
	Done := FALSE;
	IF NOT Execute THEN
		uiFbState := 0;
		Error := FALSE;
		ErrorID := 0;
	END_IF

END_CASE

END_FUNCTION_BLOCK

// POUs/LinMot MC Function Blocks Advanced/LMav_PStream
FUNCTION_BLOCK LMav_PStream
VAR_INPUT
	Enable 			:BOOL;	(*Enable P streaming*)
	Position		:REAL;	(*Setpoint Position in [mm]*)
END_VAR
VAR_IN_OUT
	Axis 			:tstLM_Axis; (*Axis*)
END_VAR
VAR_OUTPUT
	Streaming 		:BOOL;	(*Streaming / FB Busy*)
	Error 			:BOOL;	(*Error detected*)
	ErrorID			:UINT;	(*Error ID:
							01h: Axis not ready
 							02h: Axis already has command running
 							03h: Axis has error
 							04h: Command interrupted
 							05h: Command aborted
							06h: Invalid input(s)
							*)
END_VAR
VAR
	uiCState		:UINT;	(*internal -> *)
	uiFbState 		:UINT;	(*internal -> *)
	rTrig 			:LM_R_TRIG;	(*internal -> *)
	udiTmpDWord		:UDINT;	(*internal -> *)
	bTemp			:BOOL;	(*internal -> *)

	uiCmdHeader 	:UINT := 16#0300; (*internal -> CommandHeader (030xh) of the "P Stream With Slave Generated Time Stamp (030xh)" motion command*)
END_VAR
(*Version history:
Date         	 | Version    		| Created under     	| Author          	| Remark 
------------------------------------------------------------------------------------------------------------------------------- 
2011-jul-20   	 | 1.0.0      		| V2.11.0 (Build 1016)	| fj  				| initial release
2011-sep-13   	 | 1.0.1      		| V2.11.0 (Build 1016)	| fj  				| removed check for "StandStill_LM" on Enable rising edge
2011-dec-01   	 | 1.0.2      		| V2.11.0 (Build 1016)	| fj  				| code optimisation
2012-apr-25   	 | 1.1.0     		| V2.11.0 (Build 1016)	| fj  				| added input parameters check
*)

(*Variablen ][ variables*)
uiCState := SHR(Axis.DrvToPlc.StateVar, 8);

(*Flankenerkennung am Execute Eingang*)
(*Edge detection on Execute input*)
rTrig(CLK:=Enable);
IF rTrig.Q AND uiCState = 16#08 AND NOT Axis.CommandRunning THEN (*Start command*)
	Axis.CommandRunning := TRUE;
	uiFbState := 1;
ELSIF rTrig.Q AND uiCState <> 16#08 THEN (*Axis not ready*)
	uiFbState := 50; (*Error state*)
	Error := TRUE;
	ErrorID := 16#01; (*Axis not ready*)
ELSIF rTrig.Q AND Axis.CommandRunning THEN (*Axis already has a command running*)
	uiFbState := 50; (*Error state*)
	Error := TRUE;
	ErrorID := 16#02; (*Axis already has a command running*)
END_IF

IF Streaming AND uiCState = 16#04 THEN
	Axis.CommandRunning := FALSE;
	uiFbState := 50;
	Error := TRUE;
	ErrorID := 16#03; (*Axis has error*)
END_IF

IF Streaming AND uiCState <> 16#08 THEN
	Axis.CommandRunning := FALSE;
	uiFbState := 50; (*Error state*)
	Error := TRUE;
	ErrorID := 16#04; (*Command interupted*)
ELSIF Streaming AND Axis.CommandAborted THEN
	uiFbState := 50; (*Error state*)
	Error := TRUE;
	ErrorID := 16#05; (*Command aborted*)
END_IF

(*uiState machine*)
CASE uiFbState OF
	0:	;

	1:	(*Check inputs on valid value*)
		IF (-214748.0 <= Position AND Position <= 214748.0)
			THEN
			(*Streaming*)
			bTemp := Axis.PlcToDrv.MCHeader.0;
			Axis.PlcToDrv.MCHeader := uiCmdHeader;
			Axis.PlcToDrv.MCHeader.0 := NOT bTemp;

			(*Parameter Umrechung*)
			(*Calculate parameters*)
			udiTmpDWord := DINT_TO_UDINT(REAL_TO_DINT(Position * 10000)); (*Position*)
			Axis.PlcToDrv.MCParaWord0 := UDINT_TO_UINT(udiTmpDWord);
			Axis.PlcToDrv.MCParaWord1 := UDINT_TO_UINT(ROR(udiTmpDWord,16));

			LM_UptMCI(Axis);

			Streaming := TRUE;
		
			IF NOT Enable THEN
				uiFbState := 2;
			END_IF
		ELSE
			Axis.CommandRunning := FALSE;
			uiFbState := 50; (*Error state*)
			Error := TRUE;
			ErrorID := 16#06; (*Invalid input(s)*)
		END_IF

	2:	(*Stop streaming*)
		bTemp := Axis.PlcToDrv.MCHeader.0;
		Axis.PlcToDrv.MCHeader := 16#03F0; (*Header 03F0h (Stop Stream)*)
		Axis.PlcToDrv.MCHeader.0 := NOT bTemp;

		uiFbState := 3;

	3:	IF Axis.PlcToDrv.MCHeader.0 = Axis.DrvToPlc.StateVar.0 THEN
			Streaming := FALSE;
			Axis.PlcToDrv.MCHeader := 16#0000; (*No Operation*)
			Axis.PlcToDrv.MCHeader.0 := Axis.DrvToPlc.StateVar.0;
			Axis.CommandRunning := FALSE;
			uiFbState := 0;
		END_IF

	50:	Error := TRUE;
		Axis.PlcToDrv.MCHeader := 16#0000; (*No Operation*)
		Streaming := FALSE;
		uiFbState := 51;

	51:	 IF NOT Enable THEN
			uiFbState := 0;
			Error := FALSE;
			ErrorID := 0;
		END_IF

END_CASE

END_FUNCTION_BLOCK

// POUs/LinMot MC Function Blocks Advanced/LMav_PVStream
FUNCTION_BLOCK LMav_PVStream
VAR_INPUT
	Enable 			:BOOL;	(*Enable PV streaming*)
	Position		:REAL;	(*Setpoint position in [mm]*)
	Velocity		:REAL;	(*Setpoint velocity in [mm/s]*)
END_VAR
VAR_IN_OUT
	Axis 			:tstLM_Axis; (*Axis*)
END_VAR
VAR_OUTPUT
	Streaming 		:BOOL;	(*Streaming / FB Busy*)
	Error 			:BOOL;	(*Error detected*)
	ErrorID			:UINT;	(*Error ID:
							01h: Axis not ready
 							02h: Axis already has command running
 							03h: Axis has error
 							04h: Command interrupted
 							05h: Command aborted
							06h: Invalid input(s)
							*)
END_VAR
VAR
	uiCState		:UINT;	(*internal -> *)
	uiFbState 		:UINT;	(*internal -> *)
	rTrig 			:LM_R_TRIG;	(*internal -> *)
	udiTmpDWord		:UDINT;	(*internal -> *)
	bTemp			:BOOL;	(*internal -> *)

	uiCmdHeader 	:UINT := 16#0310; (*internal -> CommandHeader (031xh) of the "PV Stream With Slave Generated Time Stamp (031xh)" motion command*)
END_VAR
(*Version history:
Date         	 | Version    		| Created under     	| Author          	| Remark 
------------------------------------------------------------------------------------------------------------------------------- 
2011-jul-20   	 | 1.0.0      		| V2.11.0 (Build 1016)	| fj  				| initial release
2011-sep-13   	 | 1.0.1      		| V2.11.0 (Build 1016)	| fj  				| removed check for "StandStill_LM" on Enable rising edge
2011-dec-01   	 | 1.0.2      		| V2.11.0 (Build 1016)	| fj  				| code optimisation
2012-apr-25   	 | 1.1.0     		| V2.11.0 (Build 1016)	| fj  				| added input parameters check
*)

(*Variablen ][ variables*)
uiCState := SHR(Axis.DrvToPlc.StateVar, 8);

(*Flankenerkennung am Execute Eingang*)
(*Edge detection on Execute input*)
rTrig(CLK:=Enable);
IF rTrig.Q AND uiCState = 16#08 AND NOT Axis.CommandRunning THEN (*Start command*)
	Axis.CommandRunning := TRUE;
	uiFbState := 1;
ELSIF rTrig.Q AND uiCState <> 16#08 THEN (*Axis not ready*)
	uiFbState := 50; (*Error state*)
	Error := TRUE;
	ErrorID := 16#01; (*Axis not ready*)
ELSIF rTrig.Q AND Axis.CommandRunning THEN (*Axis already has a command running*)
	uiFbState := 50; (*Error state*)
	Error := TRUE;
	ErrorID := 16#02; (*Axis already has a command running*)
END_IF

IF Streaming AND uiCState = 16#04 THEN
	Axis.CommandRunning := FALSE;
	uiFbState := 50;
	Error := TRUE;
	ErrorID := 16#03; (*Axis has error*)
END_IF

IF Streaming AND uiCState <> 16#08 THEN
	Axis.CommandRunning := FALSE;
	uiFbState := 50; (*Error state*)
	Error := TRUE;
	ErrorID := 16#04; (*Command interupted*)
ELSIF Streaming AND Axis.CommandAborted THEN
	uiFbState := 50; (*Error state*)
	Error := TRUE;
	ErrorID := 16#05; (*Command aborted*)
END_IF

(*uiState machine*)
CASE uiFbState OF
	0:	;

	1:	(*Check inputs on valid value*)
		IF (-214748.0 <= Position AND Position <= 214748.0)
			AND (-2147.0 <= Velocity AND Velocity <= 2147.0)
			THEN
			(*Streaming*)
			bTemp := Axis.PlcToDrv.MCHeader.0;
			Axis.PlcToDrv.MCHeader := uiCmdHeader;
			Axis.PlcToDrv.MCHeader.0 := NOT bTemp;

			(*Parameter Umrechung*)
			(*Calculate parameters*)
			udiTmpDWord := DINT_TO_UDINT(REAL_TO_DINT(Position * 10000)); (*Position*)
			Axis.PlcToDrv.MCParaWord0 := UDINT_TO_UINT(udiTmpDWord);
			Axis.PlcToDrv.MCParaWord1 := UDINT_TO_UINT(ROR(udiTmpDWord,16));

			udiTmpDWord := DINT_TO_UDINT(REAL_TO_DINT(Velocity * 1000)); (*Velocity*)
			Axis.PlcToDrv.MCParaWord2 := UDINT_TO_UINT(udiTmpDWord);
			Axis.PlcToDrv.MCParaWord3 := UDINT_TO_UINT(ROR(udiTmpDWord,16));

			LM_UptMCI(Axis);

			Streaming := TRUE;
		
			IF NOT Enable THEN
				uiFbState := 2;
			END_IF
		ELSE
			Axis.CommandRunning := FALSE;
			uiFbState := 50; (*Error state*)
			Error := TRUE;
			ErrorID := 16#06; (*Invalid input(s)*)
		END_IF

	2:	(*Stop streaming*)
		bTemp := Axis.PlcToDrv.MCHeader.0;
		Axis.PlcToDrv.MCHeader := 16#03F0; (*Header 03F0h (Stop Stream)*)
		Axis.PlcToDrv.MCHeader.0 := NOT bTemp;

		uiFbState := 3;

	3:	IF Axis.PlcToDrv.MCHeader.0 = Axis.DrvToPlc.StateVar.0 THEN
			Streaming := FALSE;
			Axis.PlcToDrv.MCHeader := 16#0000; (*No Operation*)
			Axis.PlcToDrv.MCHeader.0 := Axis.DrvToPlc.StateVar.0;
			Axis.CommandRunning := FALSE;
			uiFbState := 0;
		END_IF

	50:	Error := TRUE;
		Axis.PlcToDrv.MCHeader := 16#0000; (*No Operation*)
		Streaming := FALSE;
		uiFbState := 51;

	51:	 IF NOT Enable THEN
			uiFbState := 0;
			Error := FALSE;
			ErrorID := 0;
		END_IF

END_CASE

END_FUNCTION_BLOCK

// POUs/LinMot MC Function Blocks Advanced/LMav_RunCurve
FUNCTION_BLOCK LMav_RunCurve
VAR_INPUT
	Execute			:BOOL;	(*Execute command)*)
	CurveID			:UINT;	(*Curve ID*)
	CurveOffset		:REAL;	(*Offset in [mm]*)
	TimeScale		:REAL;	(*Time scale (0-200%)*)
	AmplitudeScale	:REAL;	(*Amplitude scale (-2000% to +2000%*)
END_VAR
VAR_IN_OUT
	Axis 			:tstLM_Axis; (*Axis*)
END_VAR
VAR_OUTPUT
	Done			:BOOL;	(*Command has been executed*)
	Busy			:BOOL;	(*Command running / FB Busy*)
	Error			:BOOL;	(*Error detected*)
	ErrorID			:UINT;	(*Error ID:
							01h: Axis not ready
 							02h: Axis already has command running
 							03h: Axis has error
 							04h: Command interrupted
 							05h: Command aborted
							06h: Invalid input(s)
							*)
END_VAR
VAR
	usiOldCmdCount 	:USINT;	(*internal -> *)
	usiNewCmdCount	:USINT;	(*internal -> *)
	uiCState		:UINT;	(*internal -> *)
	uiFbState		:UINT;	(*internal -> *)
	rTrig			:LM_R_TRIG;	(*internal -> *)
	udiTmpDWord		:UDINT;	(*internal -> *)

 	uiCmdHeader 	:UINT := 16#0440;	(*CommandHeader (044xh) of the "Time Curve With Adjustable Offset, Time Scale & Amplitude Scale (044xh)" motion command*)
END_VAR
(*Version history:
Date         	 | Version    		| Created under     	| Author          	| Remark 
------------------------------------------------------------------------------------------------------------------------------- 
2011-jul-12   	 | 1.0.0      		| V2.11.0 (Build 1016)	| fj  				| initial release
2011-sep-13   	 | 1.0.1      		| V2.11.0 (Build 1016)	| fj  				| removed check for "StandStill_LM" on Execute rising edge
2011-dec-01   	 | 1.0.2      		| V2.11.0 (Build 1016)	| fj  				| code optimisation
2012-apr-25   	 | 1.1.0     		| V2.11.0 (Build 1016)	| fj  				| added input parameters check
*)

(*Variablen ][ variables*)
usiOldCmdCount := SHR(UINT_TO_USINT(SHL(Axis.DrvToPlc.StateVar,4)),4);
uiCState := SHR(Axis.DrvToPlc.StateVar, 8);

(*Flankenerkennung am Execute Eingang*)
(*Edge detection on Execute input*)
rTrig(CLK:=Execute);
IF rTrig.Q AND uiCState = 16#08 AND NOT Axis.CommandRunning THEN (*Start command*)
	Axis.CommandRunning := TRUE;
	Busy := TRUE;
	uiFbState := 1;
ELSIF rTrig.Q AND Busy THEN (*Restart command / New rising edge on execute input*)
	Axis.CommandRunning := TRUE;
	Busy := TRUE;
	uiFbState := 1;
ELSIF rTrig.Q AND uiCState <> 16#08 THEN (*Axis not ready*)
	uiFbState := 50; (*Error state*)
	Error := TRUE;
	ErrorID := 16#01; (*Axis not ready*)
ELSIF rTrig.Q AND Axis.CommandRunning AND NOT Busy THEN (*Axis already has a command running*)
	uiFbState := 50; (*Error state*)
	Error := TRUE;
	ErrorID := 16#02; (*Axis already has a command running*)
END_IF

IF Busy AND uiCState = 16#04 THEN
	Axis.CommandRunning := FALSE;
	uiFbState := 50;
	Error := TRUE;
	ErrorID := 16#03; (*Axis has error*)
END_IF

IF Busy AND uiCState <> 16#08 THEN
	Axis.CommandRunning := FALSE;
	uiFbState := 50; (*Error state*)
	Error := TRUE;
	ErrorID := 16#04; (*Command interupted*)
ELSIF Busy AND Axis.CommandAborted THEN
	uiFbState := 50; (*Error state*)
	Error := TRUE;
	ErrorID := 16#05; (*Command aborted*)
END_IF

(*State machine*)
CASE uiFbState OF
	0:	;

	1:	(*Check inputs on valid value*)
		IF (1 <= CurveID AND CurveID <= 255)
			AND (-214748.0 <= CurveOffset AND CurveOffset <= 214748.0)
			AND (0.0 < TimeScale AND TimeScale <= 200.0)
			AND (-2000.0 <= AmplitudeScale AND AmplitudeScale <= 2000.0)
			THEN
			(*Befehlskopf mit CMD Count berechen und senden ][ Calculate and send command header*)
			usiNewCmdCount := (usiOldCmdCount + 1) MOD 16 ; (*MOD 16*)
			Axis.PlcToDrv.MCHeader := 16#0000; (*Reset Header*)
			Axis.PlcToDrv.MCHeader := uiCmdHeader + usiNewCmdCount;

			Axis.PlcToDrv.MCParaWord0 := CurveID; (*CurveID*)

			udiTmpDWord := DINT_TO_UDINT(REAL_TO_DINT(CurveOffset * 10000)); (*Curve Offset*)
			Axis.PlcToDrv.MCParaWord1 := UDINT_TO_UINT(udiTmpDWord);
			Axis.PlcToDrv.MCParaWord2 := UDINT_TO_UINT(ROR(udiTmpDWord,16));

			Axis.PlcToDrv.MCParaWord3 := REAL_TO_UINT(TimeScale * 100); (*Time Scale*)
			Axis.PlcToDrv.MCParaWord4 := REAL_TO_UINT(AmplitudeScale * 10); (*Amplitude Scale*)

			LM_UptMCI(Axis);

			uiFbState := 2;
		ELSE
			Axis.CommandRunning := FALSE;
			uiFbState := 50; (*Error state*)
			Error := TRUE;
			ErrorID := 16#06; (*Invalid input(s)*)
		END_IF

	2:	(*Prüfen ob Befehl ausgeführt ][ Check if command has been executed*)
		IF usiOldCmdCount = usiNewCmdCount AND uiCState = 16#08 AND Axis.DrvToPlc.StateVar.6 THEN
			Done := TRUE;
			Busy := FALSE;
			Axis.PlcToDrv.MCHeader := 16#0000 + usiNewCmdCount; (*Send no operation*)
			Axis.CommandRunning := FALSE;
			uiFbState := 3;
		END_IF

	3:	IF NOT Execute THEN
			uiFbState := 0;
			Busy := FALSE;
			Done := FALSE;
		END_IF

	50:	Error := TRUE;
		Busy := FALSE;
		Done := FALSE;
		IF NOT Execute THEN
			uiFbState := 0;
			Error := FALSE;
			ErrorID := 0;
		END_IF

END_CASE

END_FUNCTION_BLOCK

// POUs/Rotary Motors/LMct_RotaryMotorControl
FUNCTION_BLOCK LMct_RotaryMotorControl
VAR_INPUT
	SwitchOn		    :BOOL;	(*Switch on motor*)
	Home				:BOOL;	(*Start homing procedure*)
	ErrorAcknowledge	:BOOL;	(*Error acknowledge*)
	JogPlus				:BOOL;	(*Jog move postive*)
	JogMinus			:BOOL;	(*Jog move negative*)
	SetReference		:BOOL;	(*Set rotary motor reference*)
	ReferenceAngle		:DINT;	(*[Units]*)
	ModuloFactor		:DINT;	(*[Units]*)
END_VAR
VAR_IN_OUT
	Axis	       		:tstLM_Axis; (*Axis reference*)
END_VAR
VAR_OUTPUT
	OperationEnabled	:BOOL;	(*Axis powered on*)
	SwitchOnLocked		:BOOL;	(*Switch on locked*)
	Homed     	      	:BOOL;	(*Axis has reference*)
	ReferenceSet		:BOOL;	(*Reference Set*)
	MotionActive		:BOOL;	(*Motion active (Setpoint generation (VAI, curve) active)*)
	Jogging				:BOOL;	(*Axis is moving in jog mode*)
	Warning         	:BOOL;	(*Warning detected*)
	Error          		:BOOL;	(*Error detected*)
	ErrorCode      		:UINT;	(*Error code, see MotionCtrlSW manual*)
	MotorDemandAngle  	:DINT;	(*Demand angle in [Units]*)
	MotorActualAngle  	:DINT;	(*Actual position in [Units]*)
	NrOfRevolutions		:DINT;	(*Number of revolutions*)
	ActualCurrent   	:REAL;	(*Actual motor current in [A]*)
END_VAR
VAR
	uiState        		:UINT;	(*internal -> Current state of the drive*)
	rTrigHome 			:LM_R_TRIG;	(*internal ->*)
	fTrigHome 			:LM_F_TRIG;	(*internal ->*)
	rTrigSetReference	:LM_R_TRIG;	(*internal ->*)
	dOldMotorDemandAngle:DINT;	(*internal ->*)
END_VAR
(*Version history:
Date         	 | Version    		| Created under     	| Author          	| Remark 
------------------------------------------------------------------------------------------------------------------------------- 
2014-oct-20   	 | 1.0.0.0     		| v3.1.4014.0			| fj  				| initial version
2015-feb-04   	 | 1.0.0.1     		| v3.1.4014.0			| fj  				| avoid demand angle == modulo factor -> set demand angle to 0
*)

(*Eingänge zuweisen/lesen ][ Read and allocate inputs*)
	(*Calculate motor demand angle and number of revolutions*)
	MotorDemandAngle := MotorDemandAngle + (Axis.DrvToPlc.ComDemandPosition - dOldMotorDemandAngle);
	dOldMotorDemandAngle := Axis.DrvToPlc.ComDemandPosition;
	IF MotorDemandAngle < 0 THEN
		MotorDemandAngle := MotorDemandAngle + ModuloFactor;
		IF NrOfRevolutions = -2147483648 THEN //Prevent DINT underflow
			NrOfRevolutions := 2147483647;
		ELSE
			NrOfRevolutions := NrOfRevolutions - 1;
		END_IF;
	ELSIF MotorDemandAngle > ModuloFactor THEN
		MotorDemandAngle := MotorDemandAngle - ModuloFactor;
		IF NrOfRevolutions = 2147483647 THEN //Prevent DINT overflow
			NrOfRevolutions := -2147483648;
		ELSE
			NrOfRevolutions := NrOfRevolutions + 1;
		END_IF;
	ELSIF MotorDemandAngle = ModuloFactor THEN  (*If the demand angle is exactly the modulo factor set demand angle to 0*)
		MotorDemandAngle :=0;
		IF NrOfRevolutions = 2147483647 THEN (*Prevent DINT overflow*)
			NrOfRevolutions := -2147483648;
		ELSE
			NrOfRevolutions := NrOfRevolutions + 1;
		END_IF;
	END_IF;

	(*Calculate motor actual angle*)
	MotorActualAngle := MotorDemandAngle - (Axis.DrvToPlc.ComDemandPosition - Axis.DrvToPlc.ComActualPosition);
	IF MotorActualAngle < 0 THEN
		MotorActualAngle := MotorActualAngle + ModuloFactor;
	ELSIF MotorActualAngle > ModuloFactor THEN
		MotorActualAngle := MotorActualAngle - ModuloFactor;
	END_IF;

	(*Workaround for different XML current definitions (16Bit/32Bit)*)
	IF Axis.DrvToPlc.ComActualCurrent32 = 0 AND Axis.DrvToPlc.ComActualCurrent16 = 0 THEN
		ActualCurrent := 0;
	ELSIF Axis.DrvToPlc.ComActualCurrent32 <> 0 AND Axis.DrvToPlc.ComActualCurrent16 = 0 THEN
		ActualCurrent := DINT_TO_REAL(Axis.DrvToPlc.ComActualCurrent32)/1000;
	ELSIF Axis.DrvToPlc.ComActualCurrent32 = 0 AND Axis.DrvToPlc.ComActualCurrent16 <> 0 THEN
		ActualCurrent := INT_TO_REAL(Axis.DrvToPlc.ComActualCurrent16)/1000;
	ELSE
		ActualCurrent := DINT_TO_REAL(Axis.DrvToPlc.ComActualCurrent32)/1000; (*If both 16/32Bit currents aren't 0 32Bit has higher priority*)
	END_IF

(*Variablen ][ variables*)
	uiState := SHR(Axis.DrvToPlc.StateVar, 8);
	SwitchOnLocked := Axis.DrvToPlc.StatusWord.6;
	Warning := Axis.DrvToPlc.StatusWord.7;
	MotionActive := Axis.DrvToPlc.StatusWord.13;
	OperationEnabled := Axis.DrvToPlc.StatusWord.0;

(*=============================================================================
*  State Machine
===============================================================================*)    

CASE uiState OF
	(*Not Ready to Switch On*)
	00:	Axis.AxisState := Disabled_LM;

	(*State 4: Error*)
	04:	ErrorCode := UINT_TO_USINT(Axis.DrvToPlc.StateVar);
		Error := TRUE;
		Axis.AxisState := ErrorStop_LM;

	(*State 8: Operation Enabled*)
	08:	Homed := Axis.DrvToPlc.StateVar.7;
		IF Axis.DrvToPlc.StatusWord.13 AND NOT (Axis.AxisState = Stopping_LM) THEN
			Axis.AxisState := DiscreteMotion_LM;
		ELSIF NOT Axis.DrvToPlc.StatusWord.13 AND NOT (Axis.AxisState = Stopping_LM) THEN
			Axis.AxisState := StandStill_LM;
		END_IF

	(*State 9: Homing*)
	09:	Axis.AxisState := Homing_LM;
		IF Axis.DrvToPlc.StateVar = 16#090F THEN
            ReferenceSet := TRUE;
            IF ModuloFactor > 0 THEN (*prevent division by 0*)
                NrOfRevolutions := (ReferenceAngle - (ReferenceAngle MOD ModuloFactor)) / ModuloFactor;
            END_IF;
            MotorDemandAngle := ReferenceAngle MOD ModuloFactor;
            MotorActualAngle := MotorDemandAngle - (Axis.DrvToPlc.ComDemandPosition - Axis.DrvToPlc.ComActualPosition); (*Act angle = demand angle - position error*)
            IF MotorActualAngle < 0 THEN
                MotorActualAngle := MotorActualAngle + ModuloFactor;
            ELSIF MotorActualAngle > ModuloFactor THEN
                MotorActualAngle := MotorActualAngle - ModuloFactor;
            END_IF;
            Axis.PlcToDrv.ControlWord.11 := FALSE;
        END_IF;

	(*State 14: Error Behaviour QuickStop*)
	14:	Axis.AxisState := ErrorStop_LM;

	(*State 16: Jogging +*)
	16:	Axis.AxisState := Jogging_LM;

	(*State 17: Jogging -*)
	17:	Axis.AxisState := Jogging_LM;

END_CASE;


(*Wenn der drive nicht im Fehlerzustand ist, werden Error und ErrorCode auf Null gesetzt*)
(*If the drive is not in Error state, Error and ErrorCode are set to zero*)
IF uiState <> 16#04 THEN
	Error := FALSE;
	ErrorCode := 16#00;
END_IF;

IF uiState <> 16#08 THEN
	Axis.PlcToDrv.MCHeader := 16#0000; (*Reset Header to prevent "MC Cmd in wrong state" error*)
	Axis.CommandRunning := FALSE;
	Axis.CommandAborted := FALSE;
END_IF;

(*Switch On*)
Axis.PlcToDrv.ControlWord.0 := SwitchOn;
IF NOT Axis.PlcToDrv.ControlWord.0 AND NOT (uiState = 4 OR uiState = 14) THEN
	Axis.AxisState := Disabled_LM;
END_IF

(*Set Reference*)
rTrigSetReference(CLK:=SetReference);
IF rTrigSetReference.Q THEN
    ReferenceSet := TRUE;
    IF ModuloFactor > 0 THEN (*prevent division by 0*)
        NrOfRevolutions := (ReferenceAngle - (ReferenceAngle MOD ModuloFactor)) / ModuloFactor;
    END_IF;
    
    MotorDemandAngle := ReferenceAngle MOD ModuloFactor;
    IF MotorDemandAngle < 0 THEN
        MotorDemandAngle := MotorDemandAngle + ModuloFactor;
    ELSIF MotorDemandAngle > ModuloFactor THEN
        MotorDemandAngle := MotorDemandAngle - ModuloFactor;
    END_IF;

    MotorActualAngle := MotorDemandAngle - (Axis.DrvToPlc.ComDemandPosition - Axis.DrvToPlc.ComActualPosition); (*Istwinkel = Sollwinkel - Schleppfehler*)
    IF MotorActualAngle < 0 THEN
        MotorActualAngle := MotorActualAngle + ModuloFactor;
    ELSIF MotorActualAngle > ModuloFactor THEN
        MotorActualAngle := MotorActualAngle - ModuloFactor;
    END_IF;
END_IF;

(*Home*)
rTrigHome(CLK:=Home);
fTrigHome(CLK:=Home);
IF rTrigHome.Q THEN
	Axis.PlcToDrv.ControlWord.11 := TRUE;
END_IF
IF fTrigHome.Q  THEN
	Axis.PlcToDrv.ControlWord.11 := FALSE;
END_IF

IF uiState = 16#09 OR (Axis.PlcToDrv.ControlWord.11 AND NOT (uistate = 16#09)) THEN
	Homed := FALSE;
ELSE
	Homed := Axis.DrvToPlc.StatusWord.11;
END_IF

(*Error acknowledge*)
Axis.PlcToDrv.ControlWord.7 := ErrorAcknowledge;

(*JogPlus*)
Axis.PlcToDrv.ControlWord.8 := JogPlus;

(*JogMinus*)
Axis.PlcToDrv.ControlWord.9 := JogMinus;

IF (uiState = 16 OR uiState = 17) AND UINT_TO_USINT(Axis.DrvToPlc.StateVar) = 16#01 THEN
	Jogging := TRUE;
ELSE
	Jogging := FALSE;
END_IF

END_FUNCTION_BLOCK

// POUs/Rotary Motors/LMmt_RotIncrActAngle
FUNCTION_BLOCK LMmt_RotIncrActAngle
VAR_INPUT
	Execute			:BOOL;	(*Execute command*)
	Distance		:DINT;	(*Distance in [Units]*)
	Velocity		:REAL;	(*[Units/s]*)
	Acceleration	:REAL;	(*[Units/s^2]*)
	Deceleration	:REAL;	(*[Units/s^2]*)
END_VAR
VAR_IN_OUT
	Axis			:tstLM_Axis; (*Axis reference*)
END_VAR
VAR_OUTPUT
	Done			:BOOL;	(*Command has been executed*)
	Busy			:BOOL;	(*Command running / FB Busy*)
	Error			:BOOL;	(*Error detected*)
	ErrorID			:UINT;	(*Error ID:
							01h: Axis not ready
 							02h: Axis already has command running
 							03h: Axis has error
 							04h: Command interrupted
 							05h: Command aborted
							06h: Invalid input(s)
							*)
END_VAR
VAR
	usiOldCmdCount 	:USINT;	(*internal -> *)
	usiNewCmdCount	:USINT;	(*internal -> *)
	uiCState		:UINT;	(*internal -> *)
	uiFbState		:UINT;	(*internal -> *)
	rTrig			:LM_R_TRIG;	(*internal -> *)
	udiTmpDWord		:UDINT;	(*internal -> *)

 	uiCmdHeader 	:UINT := 16#0150;	(*CommandHeader (015xh) of the "VAI Increment Act Position (015xh)" motion command*)
END_VAR
(*Version history:
Date         	 | Version    		| Created under     	| Author          	| Remark 
------------------------------------------------------------------------------------------------------------------------------- 
2014-oct-20   	 | 1.0.0.0     		| v3.1.4014.0			| fj  				| initial version
*)

(*Variablen ][ variables*)
usiOldCmdCount := SHR(UINT_TO_USINT(SHL(Axis.DrvToPlc.StateVar,4)),4);
uiCState := SHR(Axis.DrvToPlc.StateVar, 8);

(*Flankenerkennung am Execute Eingang*)
(*Edge detection on Execute input*)
rTrig(CLK:=Execute);
IF rTrig.Q AND uiCState = 16#08 AND NOT Axis.CommandRunning THEN (*Start command*)
	Axis.CommandRunning := TRUE;
	Busy := TRUE;
	uiFbState := 1;
ELSIF rTrig.Q AND Busy THEN (*Restart command / New rising edge on execute input*)
	Axis.CommandRunning := TRUE;
	Busy := TRUE;
	uiFbState := 1;
ELSIF rTrig.Q AND uiCState <> 16#08 THEN (*Axis not ready*)
	uiFbState := 50; (*Error state*)
	Error := TRUE;
	ErrorID := 16#01; (*Axis not ready*)
ELSIF rTrig.Q AND Axis.CommandRunning AND NOT Busy THEN (*Axis already has a command running*)
	uiFbState := 50; (*Error state*)
	Error := TRUE;
	ErrorID := 16#02; (*Axis already has a command running*)
END_IF

IF Busy AND uiCState = 16#04 THEN
	Axis.CommandRunning := FALSE;
	uiFbState := 50;
	Error := TRUE;
	ErrorID := 16#03; (*Axis has error*)
END_IF

IF Busy AND uiCState <> 16#08 THEN
	Axis.CommandRunning := FALSE;
	uiFbState := 50; (*Error state*)
	Error := TRUE;
	ErrorID := 16#04; (*Command interupted*)
ELSIF Busy AND Axis.CommandAborted THEN
	uiFbState := 50; (*Error state*)
	Error := TRUE;
	ErrorID := 16#05; (*Command aborted*)
END_IF

(*State machine*)
CASE uiFbState OF
    0:  ;
        
    1:  (*Check inputs on valid value*)
        IF (-2147483648 < Distance AND Distance < 2147483647)
            AND (0.0 < Velocity)
            AND (0.0 < Acceleration)
            AND (0.0 < Deceleration)
        THEN
        (*Befehlskopf mit CMD Count berechen und senden ][ Calculate and send command header*)
            usiNewCmdCount := (usiOldCmdCount + 1) MOD 16; (*Command counter MOD 16*)
            Axis.PlcToDrv.MCHeader := 16#0000; (*Reset Header*)
            Axis.PlcToDrv.MCHeader := uiCmdHeader + usiNewCmdCount;
                      
			udiTmpDWord := DINT_TO_UDINT(Distance); (*Position increment*)
            Axis.PlcToDrv.MCParaWord0 := UDINT_TO_UINT(udiTmpDWord);
            Axis.PlcToDrv.MCParaWord1 := UDINT_TO_UINT(ROR(udiTmpDWord, 16));
            
            udiTmpDWord := DINT_TO_UDINT(REAL_TO_DINT(Velocity / 10)); (*Velocity*)
            Axis.PlcToDrv.MCParaWord2 := UDINT_TO_UINT(udiTmpDWord);
            Axis.PlcToDrv.MCParaWord3 := UDINT_TO_UINT(ROR(udiTmpDWord, 16));
            
            udiTmpDWord := DINT_TO_UDINT(REAL_TO_DINT(Acceleration / 100)); (*Acceleration*)
            Axis.PlcToDrv.MCParaWord4 := UDINT_TO_UINT(udiTmpDWord);
            Axis.PlcToDrv.MCParaWord5 := UDINT_TO_UINT(ROR(udiTmpDWord, 16));
            
            udiTmpDWord := DINT_TO_UDINT(REAL_TO_DINT(Deceleration / 100)); (*Deceleration*)
            Axis.PlcToDrv.MCParaWord6 := UDINT_TO_UINT(udiTmpDWord);
            Axis.PlcToDrv.MCParaWord7 := UDINT_TO_UINT(ROR(udiTmpDWord, 16));
			
			LM_UptMCI(Axis);
            
            uiFbState := 2;
        ELSE
            Axis.CommandRunning := FALSE;
            uiFbState := 50; (*Error state*)
            Error := TRUE;
            ErrorID := 16#06; (*Invalid input(s)*)
        END_IF;
        
    2:  (*Prüfen ob Befehl ausgeführt ][ Check if command has been executed*)
        IF usiOldCmdCount = usiNewCmdCount AND uiCState = 16#08 AND Axis.DrvToPlc.StateVar.6 THEN
            Done := TRUE;
            Busy := FALSE;
            Axis.PlcToDrv.MCHeader := 16#0000 + usiNewCmdCount; (*Send no operation*)
            Axis.CommandRunning := FALSE;
            uiFbState := 3;
        END_IF;
        
    3:  IF NOT Execute THEN
            uiFbState := 0;
            Busy := FALSE;
            Done := FALSE;
        END_IF;
        
    50: Error := TRUE;
        Busy := FALSE;
        Done := FALSE;
        IF NOT Execute THEN
            uiFbState := 0;
            Error := FALSE;
            ErrorID := 0;
        END_IF;
        
END_CASE;

END_FUNCTION_BLOCK

// POUs/Rotary Motors/LMmt_RotIncrActAngleJ
FUNCTION_BLOCK LMmt_RotIncrActAngleJ
VAR_INPUT
	Execute			:BOOL;	(*Execute command*)
	Distance		:DINT;	(*Distance in [Units]*)
	Velocity		:REAL;	(*Maximal velocity [Units/s]*)
	Acceleration	:REAL;	(*Maximal acceleration [Units/s^2]*)
	Deceleration	:REAL;	(*Maximal deceleration [Units/s^2]*)
	Jerk			:REAL;	(*Jerk [Units/s^3]*)
END_VAR
VAR_IN_OUT
	Axis			:tstLM_Axis; (*Axis reference*)
END_VAR
VAR_OUTPUT
	Done			:BOOL;	(*Command has been executed*)
	Busy			:BOOL;	(*Command running / FB Busy*)
	Error			:BOOL;	(*Error detected*)
	ErrorID			:UINT;	(*Error ID:
							01h: Axis not ready
 							02h: Axis already has command running
 							03h: Axis has error
 							04h: Command interrupted
 							05h: Command aborted
							06h: Invalid input(s)
							*)
END_VAR
VAR
	usiOldCmdCount 	:USINT;	(*internal -> *)
	usiNewCmdCount	:USINT;	(*internal -> *)
	uiCState		:UINT;	(*internal -> *)
	uiFbState		:UINT;	(*internal -> *)
	rTrig			:LM_R_TRIG;	(*internal -> *)
	udiTmpDWord		:UDINT;	(*internal -> *)

 	uiCmdHeader 	:UINT := 16#3A60; (*CommandHeader (3A6xh) of the "VAJI Increment Act Pos Starting with Dem Vel = 0 and Dem Acc = 0 (3A6xh)" motion command*)
END_VAR
(*Version history:
Date         	 | Version    		| Created under     	| Author          	| Remark 
------------------------------------------------------------------------------------------------------------------------------- 
2016-jan-05    	 | 1.0.0.0     		| v3.1.4016.12			| fj  				| initial version
*)

(*Variablen ][ variables*)
usiOldCmdCount := SHR(UINT_TO_USINT(SHL(Axis.DrvToPlc.StateVar,4)),4);
uiCState := SHR(Axis.DrvToPlc.StateVar, 8);

(*Flankenerkennung am Execute Eingang*)
(*Edge detection on Execute input*)
rTrig(CLK:=Execute);
IF rTrig.Q AND uiCState = 16#08 AND NOT Axis.CommandRunning THEN (*Start command*)
	Axis.CommandRunning := TRUE;
	Busy := TRUE;
	uiFbState := 1;
ELSIF rTrig.Q AND Busy THEN (*Restart command / New rising edge on execute input*)
	Axis.CommandRunning := TRUE;
	Busy := TRUE;
	uiFbState := 1;
ELSIF rTrig.Q AND uiCState <> 16#08 THEN (*Axis not ready*)
	uiFbState := 50; (*Error state*)
	Error := TRUE;
	ErrorID := 16#01; (*Axis not ready*)
ELSIF rTrig.Q AND Axis.CommandRunning AND NOT Busy THEN (*Axis already has a command running*)
	uiFbState := 50; (*Error state*)
	Error := TRUE;
	ErrorID := 16#02; (*Axis already has a command running*)
END_IF

IF Busy AND uiCState = 16#04 THEN
	Axis.CommandRunning := FALSE;
	uiFbState := 50;
	Error := TRUE;
	ErrorID := 16#03; (*Axis has error*)
END_IF

IF Busy AND uiCState <> 16#08 THEN
	Axis.CommandRunning := FALSE;
	uiFbState := 50; (*Error state*)
	Error := TRUE;
	ErrorID := 16#04; (*Command interupted*)
ELSIF Busy AND Axis.CommandAborted THEN
	uiFbState := 50; (*Error state*)
	Error := TRUE;
	ErrorID := 16#05; (*Command aborted*)
END_IF

(*State machine*)
CASE uiFbState OF
    0:  ;
        
    1:  (*Check inputs on valid value*)
        IF (-2147483648 < Distance AND Distance < 2147483647)
            AND (0.0 < Velocity)
            AND (0.0 < Acceleration)
            AND (0.0 < Deceleration)
            AND (0.0 < Jerk AND Jerk <= 1600000000)
        THEN
        (*Befehlskopf mit CMD Count berechen und senden ][ Calculate and send command header*)
            usiNewCmdCount := (usiOldCmdCount + 1) MOD 16; (*Command counter MOD 16*)
            Axis.PlcToDrv.MCHeader := 16#0000; (*Reset Header*)
            Axis.PlcToDrv.MCHeader := uiCmdHeader + usiNewCmdCount;
                      
			udiTmpDWord := DINT_TO_UDINT(Distance); (*Position increment*)
            Axis.PlcToDrv.MCParaWord0 := UDINT_TO_UINT(udiTmpDWord);
            Axis.PlcToDrv.MCParaWord1 := UDINT_TO_UINT(ROR(udiTmpDWord, 16));
            
            udiTmpDWord := DINT_TO_UDINT(REAL_TO_DINT(Velocity / 10)); (*Velocity*)
            Axis.PlcToDrv.MCParaWord2 := UDINT_TO_UINT(udiTmpDWord);
            Axis.PlcToDrv.MCParaWord3 := UDINT_TO_UINT(ROR(udiTmpDWord, 16));
            
            udiTmpDWord := DINT_TO_UDINT(REAL_TO_DINT(Acceleration / 100)); (*Acceleration*)
            Axis.PlcToDrv.MCParaWord4 := UDINT_TO_UINT(udiTmpDWord);
            Axis.PlcToDrv.MCParaWord5 := UDINT_TO_UINT(ROR(udiTmpDWord, 16));
            
            udiTmpDWord := DINT_TO_UDINT(REAL_TO_DINT(Deceleration / 100)); (*Deceleration*)
            Axis.PlcToDrv.MCParaWord6 := UDINT_TO_UINT(udiTmpDWord);
            Axis.PlcToDrv.MCParaWord7 := UDINT_TO_UINT(ROR(udiTmpDWord, 16));
            
            udiTmpDWord := DINT_TO_UDINT(REAL_TO_DINT(Jerk) / 1000); (*Jerk*)
            Axis.PlcToDrv.MCParaWord8 := UDINT_TO_UINT(udiTmpDWord);
            Axis.PlcToDrv.MCParaWord9 := UDINT_TO_UINT(ROR(udiTmpDWord, 16));
			
			LM_UptMCI(Axis);
            
            uiFbState := 2;
        ELSE
            Axis.CommandRunning := FALSE;
            uiFbState := 50; (*Error state*)
            Error := TRUE;
            ErrorID := 16#06; (*Invalid input(s)*)
        END_IF;
        
    2:  (*Prüfen ob Befehl ausgeführt ][ Check if command has been executed*)
        IF usiOldCmdCount = usiNewCmdCount AND uiCState = 16#08 AND Axis.DrvToPlc.StateVar.6 THEN
            Done := TRUE;
            Busy := FALSE;
            Axis.PlcToDrv.MCHeader := 16#0000 + usiNewCmdCount; (*Send no operation*)
            Axis.CommandRunning := FALSE;
            uiFbState := 3;
        END_IF;
        
    3:  IF NOT Execute THEN
            uiFbState := 0;
            Busy := FALSE;
            Done := FALSE;
        END_IF;
        
    50: Error := TRUE;
        Busy := FALSE;
        Done := FALSE;
        IF NOT Execute THEN
            uiFbState := 0;
            Error := FALSE;
            ErrorID := 0;
        END_IF;
        
END_CASE;

END_FUNCTION_BLOCK

// POUs/Rotary Motors/LMmt_RotMoveAbs
FUNCTION_BLOCK LMmt_RotMoveAbs
VAR_INPUT
	Execute			:BOOL;	(*Execute command*)
	TargetAngle		:DINT;	(*Target angle in Units [0..ModuloFactor]*)
	Velocity		:REAL;	(*[Units/s]*)
	Acceleration	:REAL;	(*[Units/s^2]*)
	Deceleration	:REAL;	(*[Units/s^2]*)
	ModuloFactor	:DINT;	(*See manual*)
	MotorDemAngle	:DINT;	(*Connect from LMct_RotaryMotorControl.MotorDemandAngle*)
END_VAR
VAR_IN_OUT
	Axis			:tstLM_Axis; (*Axis reference*)
END_VAR
VAR_OUTPUT
	Done			:BOOL;	(*Command has been executed*)
	Busy			:BOOL;	(*Command running / FB Busy*)
	Error			:BOOL;	(*Error detected*)
	ErrorID			:UINT;	(*Error ID:
							01h: Axis not ready
 							02h: Axis already has command running
 							03h: Axis has error
 							04h: Command interrupted
 							05h: Command aborted
							06h: Invalid input(s)
							*)
END_VAR
VAR
	usiOldCmdCount 	:USINT;	(*internal -> *)
	usiNewCmdCount	:USINT;	(*internal -> *)
	uiCState		:UINT;	(*internal -> *)
	uiFbState		:UINT;	(*internal -> *)
	rTrig			:LM_R_TRIG;	(*internal -> *)
	udiTmpDWord		:UDINT;	(*internal -> *)

 	uiCmdHeader 	:UINT := 16#0110;	(*CommandHeader (011xh) of the "VAI Incr Dem Position (011xh)" motion command*)
END_VAR
(*Version history:
Date         	 | Version    		| Created under     	| Author          	| Remark 
------------------------------------------------------------------------------------------------------------------------------- 
2014-oct-20   	 | 1.0.0.0     		| v3.1.4014.0			| fj  				| initial version
*)

(*Variablen ][ variables*)
usiOldCmdCount := SHR(UINT_TO_USINT(SHL(Axis.DrvToPlc.StateVar,4)),4);
uiCState := SHR(Axis.DrvToPlc.StateVar, 8);

(*Flankenerkennung am Execute Eingang*)
(*Edge detection on Execute input*)
rTrig(CLK:=Execute);
IF rTrig.Q AND uiCState = 16#08 AND NOT Axis.CommandRunning THEN (*Start command*)
	Axis.CommandRunning := TRUE;
	Busy := TRUE;
	uiFbState := 1;
ELSIF rTrig.Q AND Busy THEN (*Restart command / New rising edge on execute input*)
	Axis.CommandRunning := TRUE;
	Busy := TRUE;
	uiFbState := 1;
ELSIF rTrig.Q AND uiCState <> 16#08 THEN (*Axis not ready*)
	uiFbState := 50; (*Error state*)
	Error := TRUE;
	ErrorID := 16#01; (*Axis not ready*)
ELSIF rTrig.Q AND Axis.CommandRunning AND NOT Busy THEN (*Axis already has a command running*)
	uiFbState := 50; (*Error state*)
	Error := TRUE;
	ErrorID := 16#02; (*Axis already has a command running*)
END_IF

IF Busy AND uiCState = 16#04 THEN
	Axis.CommandRunning := FALSE;
	uiFbState := 50;
	Error := TRUE;
	ErrorID := 16#03; (*Axis has error*)
END_IF

IF Busy AND uiCState <> 16#08 THEN
	Axis.CommandRunning := FALSE;
	uiFbState := 50; (*Error state*)
	Error := TRUE;
	ErrorID := 16#04; (*Command interupted*)
ELSIF Busy AND Axis.CommandAborted THEN
	uiFbState := 50; (*Error state*)
	Error := TRUE;
	ErrorID := 16#05; (*Command aborted*)
END_IF

(*State machine*)
CASE uiFbState OF
    0:  ;
        
    1:  (*Check inputs on valid value*)
        IF (0 <= TargetAngle AND TargetAngle <= ModuloFactor)
            AND (0.0 < Velocity)
            AND (0.0 < Acceleration)
            AND (0.0 < Deceleration)
            AND ModuloFactor > 0 
        THEN
        (*Befehlskopf mit CMD Count berechen und senden ][ Calculate and send command header*)
            usiNewCmdCount := (usiOldCmdCount + 1) MOD 16; (*Command counter MOD 16*)
            Axis.PlcToDrv.MCHeader := 16#0000; (*Reset Header*)
            Axis.PlcToDrv.MCHeader := uiCmdHeader + usiNewCmdCount;
                      
            IF TargetAngle > MotorDemAngle THEN
                udiTmpDWord := DINT_TO_UDINT(TargetAngle - MotorDemAngle); (*Position increment*)
            ELSIF TargetAngle < MotorDemAngle THEN
                udiTmpDWord := DINT_TO_UDINT(-1*(MotorDemAngle - TargetAngle)); (*Position increment*)
            ELSE 
                udiTmpDWord := 0; (*Position increment*)
            END_IF;
            
            Axis.PlcToDrv.MCParaWord0 := UDINT_TO_UINT(udiTmpDWord);
            Axis.PlcToDrv.MCParaWord1 := UDINT_TO_UINT(ROR(udiTmpDWord, 16));
            
            udiTmpDWord := DINT_TO_UDINT(REAL_TO_DINT(Velocity / 10)); (*Velocity*)
            Axis.PlcToDrv.MCParaWord2 := UDINT_TO_UINT(udiTmpDWord);
            Axis.PlcToDrv.MCParaWord3 := UDINT_TO_UINT(ROR(udiTmpDWord, 16));
            
            udiTmpDWord := DINT_TO_UDINT(REAL_TO_DINT(Acceleration / 100)); (*Acceleration*)
            Axis.PlcToDrv.MCParaWord4 := UDINT_TO_UINT(udiTmpDWord);
            Axis.PlcToDrv.MCParaWord5 := UDINT_TO_UINT(ROR(udiTmpDWord, 16));
            
            udiTmpDWord := DINT_TO_UDINT(REAL_TO_DINT(Deceleration / 100)); (*Deceleration*)
            Axis.PlcToDrv.MCParaWord6 := UDINT_TO_UINT(udiTmpDWord);
            Axis.PlcToDrv.MCParaWord7 := UDINT_TO_UINT(ROR(udiTmpDWord, 16));
			
			LM_UptMCI(Axis);
            
            uiFbState := 2;
        ELSE
            Axis.CommandRunning := FALSE;
            uiFbState := 50; (*Error state*)
            Error := TRUE;
            ErrorID := 16#06; (*Invalid input(s)*)
        END_IF;
        
    2:  (*Prüfen ob Befehl ausgeführt ][ Check if command has been executed*)
        IF usiOldCmdCount = usiNewCmdCount AND uiCState = 16#08 AND Axis.DrvToPlc.StateVar.6 THEN
            Done := TRUE;
            Busy := FALSE;
            Axis.PlcToDrv.MCHeader := 16#0000 + usiNewCmdCount; (*Send no operation*)
            Axis.CommandRunning := FALSE;
            uiFbState := 3;
        END_IF;
        
    3:  IF NOT Execute THEN
            uiFbState := 0;
            Busy := FALSE;
            Done := FALSE;
        END_IF;
        
    50: Error := TRUE;
        Busy := FALSE;
        Done := FALSE;
        IF NOT Execute THEN
            uiFbState := 0;
            Error := FALSE;
            ErrorID := 0;
        END_IF;
        
END_CASE;

END_FUNCTION_BLOCK

// POUs/Rotary Motors/LMmt_RotMoveAbsJ
FUNCTION_BLOCK LMmt_RotMoveAbsJ
VAR_INPUT
	Execute			:BOOL;	(*Execute command*)
	TargetAngle		:DINT;	(*Target angle in Units [0..ModuloFactor]*)
	Velocity		:REAL;	(*Maximal velocity [Units/s]*)
	Acceleration	:REAL;	(*Maximal acceleration [Units/s^2]*)
	Deceleration	:REAL;	(*Maximal deceleration [Units/s^2]*)	
	Jerk			:REAL;	(*Jerk [Units/s^3]*)
	ModuloFactor	:DINT;	(*See manual*)
	MotorDemAngle	:DINT;	(*Connect from LMct_RotaryMotorControl.MotorDemandAngle*)
END_VAR
VAR_IN_OUT
	Axis			:tstLM_Axis; (*Axis reference*)
END_VAR
VAR_OUTPUT
	Done			:BOOL;	(*Command has been executed*)
	Busy			:BOOL;	(*Command running / FB Busy*)
	Error			:BOOL;	(*Error detected*)
	ErrorID			:UINT;	(*Error ID:
							01h: Axis not ready
 							02h: Axis already has command running
 							03h: Axis has error
 							04h: Command interrupted
 							05h: Command aborted
							06h: Invalid input(s)
							*)
END_VAR
VAR
	usiOldCmdCount 	:USINT;	(*internal -> *)
	usiNewCmdCount	:USINT;	(*internal -> *)
	uiCState		:UINT;	(*internal -> *)
	uiFbState		:UINT;	(*internal -> *)
	rTrig			:LM_R_TRIG;	(*internal -> *)
	udiTmpDWord		:UDINT;	(*internal -> *)

 	uiCmdHeader 	:UINT := 16#3A10; (*CommandHeader (3A1xh) of the "VAJI Increment Dem Pos (3A1xh)" motion command*)
END_VAR
(*Version history:
Date         	 | Version    		| Created under     	| Author          	| Remark 
------------------------------------------------------------------------------------------------------------------------------- 
2016-jan-05    	 | 1.0.0.0     		| v3.1.4016.12			| fj  				| initial version
*)

(*Variablen ][ variables*)
usiOldCmdCount := SHR(UINT_TO_USINT(SHL(Axis.DrvToPlc.StateVar,4)),4);
uiCState := SHR(Axis.DrvToPlc.StateVar, 8);

(*Flankenerkennung am Execute Eingang*)
(*Edge detection on Execute input*)
rTrig(CLK:=Execute);
IF rTrig.Q AND uiCState = 16#08 AND NOT Axis.CommandRunning THEN (*Start command*)
	Axis.CommandRunning := TRUE;
	Busy := TRUE;
	uiFbState := 1;
ELSIF rTrig.Q AND Busy THEN (*Restart command / New rising edge on execute input*)
	Axis.CommandRunning := TRUE;
	Busy := TRUE;
	uiFbState := 1;
ELSIF rTrig.Q AND uiCState <> 16#08 THEN (*Axis not ready*)
	uiFbState := 50; (*Error state*)
	Error := TRUE;
	ErrorID := 16#01; (*Axis not ready*)
ELSIF rTrig.Q AND Axis.CommandRunning AND NOT Busy THEN (*Axis already has a command running*)
	uiFbState := 50; (*Error state*)
	Error := TRUE;
	ErrorID := 16#02; (*Axis already has a command running*)
END_IF

IF Busy AND uiCState = 16#04 THEN
	Axis.CommandRunning := FALSE;
	uiFbState := 50;
	Error := TRUE;
	ErrorID := 16#03; (*Axis has error*)
END_IF

IF Busy AND uiCState <> 16#08 THEN
	Axis.CommandRunning := FALSE;
	uiFbState := 50; (*Error state*)
	Error := TRUE;
	ErrorID := 16#04; (*Command interupted*)
ELSIF Busy AND Axis.CommandAborted THEN
	uiFbState := 50; (*Error state*)
	Error := TRUE;
	ErrorID := 16#05; (*Command aborted*)
END_IF

(*State machine*)
CASE uiFbState OF
    0:  ;
        
    1:  (*Check inputs on valid value*)
        IF (0 <= TargetAngle AND TargetAngle <= ModuloFactor)
            AND (0.0 < Velocity)
            AND (0.0 < Acceleration)
            AND (0.0 < Deceleration)
            AND (0.0 < Jerk AND Jerk <= 1600000000)
            AND ModuloFactor > 0 
        THEN
        (*Befehlskopf mit CMD Count berechen und senden ][ Calculate and send command header*)
            usiNewCmdCount := (usiOldCmdCount + 1) MOD 16; (*Command counter MOD 16*)
            Axis.PlcToDrv.MCHeader := 16#0000; (*Reset Header*)
            Axis.PlcToDrv.MCHeader := uiCmdHeader + usiNewCmdCount;
                      
            IF TargetAngle > MotorDemAngle THEN
                udiTmpDWord := DINT_TO_UDINT(TargetAngle - MotorDemAngle); (*Position increment*)
            ELSIF TargetAngle < MotorDemAngle THEN
                udiTmpDWord := DINT_TO_UDINT(-1*(MotorDemAngle - TargetAngle)); (*Position increment*)
            ELSE 
                udiTmpDWord := 0; (*Position increment*)
            END_IF;
            
            Axis.PlcToDrv.MCParaWord0 := UDINT_TO_UINT(udiTmpDWord);
            Axis.PlcToDrv.MCParaWord1 := UDINT_TO_UINT(ROR(udiTmpDWord, 16));
            
            udiTmpDWord := DINT_TO_UDINT(REAL_TO_DINT(Velocity / 10)); (*Velocity*)
            Axis.PlcToDrv.MCParaWord2 := UDINT_TO_UINT(udiTmpDWord);
            Axis.PlcToDrv.MCParaWord3 := UDINT_TO_UINT(ROR(udiTmpDWord, 16));
            
            udiTmpDWord := DINT_TO_UDINT(REAL_TO_DINT(Acceleration / 100)); (*Acceleration*)
            Axis.PlcToDrv.MCParaWord4 := UDINT_TO_UINT(udiTmpDWord);
            Axis.PlcToDrv.MCParaWord5 := UDINT_TO_UINT(ROR(udiTmpDWord, 16));
            
            udiTmpDWord := DINT_TO_UDINT(REAL_TO_DINT(Deceleration / 100)); (*Deceleration*)
            Axis.PlcToDrv.MCParaWord6 := UDINT_TO_UINT(udiTmpDWord);
            Axis.PlcToDrv.MCParaWord7 := UDINT_TO_UINT(ROR(udiTmpDWord, 16));
            
            udiTmpDWord := DINT_TO_UDINT(REAL_TO_DINT(Jerk) / 1000); (*Jerk*)
            Axis.PlcToDrv.MCParaWord8 := UDINT_TO_UINT(udiTmpDWord);
            Axis.PlcToDrv.MCParaWord9 := UDINT_TO_UINT(ROR(udiTmpDWord, 16));
			
			LM_UptMCI(Axis);
            
            uiFbState := 2;
        ELSE
            Axis.CommandRunning := FALSE;
            uiFbState := 50; (*Error state*)
            Error := TRUE;
            ErrorID := 16#06; (*Invalid input(s)*)
        END_IF;
        
    2:  (*Prüfen ob Befehl ausgeführt ][ Check if command has been executed*)
        IF usiOldCmdCount = usiNewCmdCount AND uiCState = 16#08 AND Axis.DrvToPlc.StateVar.6 THEN
            Done := TRUE;
            Busy := FALSE;
            Axis.PlcToDrv.MCHeader := 16#0000 + usiNewCmdCount; (*Send no operation*)
            Axis.CommandRunning := FALSE;
            uiFbState := 3;
        END_IF;
        
    3:  IF NOT Execute THEN
            uiFbState := 0;
            Busy := FALSE;
            Done := FALSE;
        END_IF;
        
    50: Error := TRUE;
        Busy := FALSE;
        Done := FALSE;
        IF NOT Execute THEN
            uiFbState := 0;
            Error := FALSE;
            ErrorID := 0;
        END_IF;
        
END_CASE;

END_FUNCTION_BLOCK

// POUs/Rotary Motors/LMmt_RotMoveInfNeg
FUNCTION_BLOCK LMmt_RotMoveInfNeg
VAR_INPUT
	Enable			:BOOL;	(*Enable command*)
	Velocity		:REAL;	(*[Units/s]*)
	Acceleration	:REAL;	(*[Units/s^2]*)
	Deceleration	:REAL;	(*[Units/s^2]*)
END_VAR
VAR_IN_OUT
	Axis			:tstLM_Axis; (*Axis reference*)
END_VAR
VAR_OUTPUT
	Done			:BOOL;	(*Command has been executed*)
	Busy			:BOOL;	(*Command running / FB Busy*)
	Error			:BOOL;	(*Error detected*)
	ErrorID			:UINT;	(*Error ID:
							01h: Axis not ready
 							02h: Axis already has command running
 							03h: Axis has error
 							04h: Command interrupted
 							05h: Command aborted
							06h: Invalid input(s)
							*)
END_VAR
VAR
	usiOldCmdCount 	:USINT;	(*internal -> *)
	usiNewCmdCount	:USINT;	(*internal -> *)
	uiCState		:UINT;	(*internal -> *)
	uiFbState		:UINT;	(*internal -> *)
	rTrig			:LM_R_TRIG;	(*internal -> *)
	udiTmpDWord		:UDINT;	(*internal -> *)

 	uiCmdHeader 	:UINT := 16#0CF0;	(*CommandHeader (0CFxh) of the "VAI Dec=Acc VAI Inifite Motion Negative Direction (0CFxh)" motion command*)
END_VAR
(*Version history:
Date         	 | Version    		| Created under     	| Author          	| Remark 
------------------------------------------------------------------------------------------------------------------------------- 
2014-oct-20   	 | 1.0.0.0     		| v3.1.4014.0			| fj  				| initial version
*)

(*Variablen ][ variables*)
usiOldCmdCount := SHR(UINT_TO_USINT(SHL(Axis.DrvToPlc.StateVar,4)),4);
uiCState := SHR(Axis.DrvToPlc.StateVar, 8);

(*Flankenerkennung am Execute Eingang*)
(*Edge detection on Execute input*)
rTrig(CLK:=Enable);
IF rTrig.Q AND uiCState = 16#08 AND NOT Axis.CommandRunning THEN (*Start command*)
	Axis.CommandRunning := TRUE;
	Busy := TRUE;
	uiFbState := 1;
ELSIF rTrig.Q AND Busy THEN (*Restart command / New rising edge on execute input*)
	Axis.CommandRunning := TRUE;
	Busy := TRUE;
	uiFbState := 1;
ELSIF rTrig.Q AND uiCState <> 16#08 THEN (*Axis not ready*)
	uiFbState := 50; (*Error state*)
	Error := TRUE;
	ErrorID := 16#01; (*Axis not ready*)
ELSIF rTrig.Q AND Axis.CommandRunning AND NOT Busy THEN (*Axis already has a command running*)
	uiFbState := 50; (*Error state*)
	Error := TRUE;
	ErrorID := 16#02; (*Axis already has a command running*)
END_IF

IF Busy AND uiCState = 16#04 THEN
	Axis.CommandRunning := FALSE;
	uiFbState := 50;
	Error := TRUE;
	ErrorID := 16#03; (*Axis has error*)
END_IF

IF Busy AND uiCState <> 16#08 THEN
	Axis.CommandRunning := FALSE;
	uiFbState := 50; (*Error state*)
	Error := TRUE;
	ErrorID := 16#04; (*Command interupted*)
ELSIF Busy AND Axis.CommandAborted THEN
	uiFbState := 50; (*Error state*)
	Error := TRUE;
	ErrorID := 16#05; (*Command aborted*)
END_IF

(*State machine*)
CASE uiFbState OF
    0:  ;
        
    1:  (*Check inputs on valid value*)
        IF (0.0 <= Velocity)
            AND (0.0 < Acceleration)
            AND (0.0 < Deceleration)
        THEN
        (*Send motion command*)
            usiNewCmdCount := (usiOldCmdCount + 1) MOD 16; (*Command counter MOD 16*)
            Axis.PlcToDrv.MCHeader := 16#0000; (*Reset Header*)
            Axis.PlcToDrv.MCHeader := uiCmdHeader + usiNewCmdCount;
            
            (*Parameter Umrechung*)
            (*Calculate parameters*)
            udiTmpDWord := REAL_TO_UDINT(Velocity / 10); (*Velocity*)
            Axis.PlcToDrv.MCParaWord0 := UDINT_TO_UINT(udiTmpDWord);
            Axis.PlcToDrv.MCParaWord1 := UDINT_TO_UINT(ROR(udiTmpDWord, 16));
            
            udiTmpDWord := REAL_TO_UDINT(Acceleration / 100); (*Acceleration*)
            Axis.PlcToDrv.MCParaWord2 := UDINT_TO_UINT(udiTmpDWord);
            Axis.PlcToDrv.MCParaWord3 := UDINT_TO_UINT(ROR(udiTmpDWord, 16));
			
			LM_UptMCI(Axis);
            
            uiFbState := 2;
        ELSE
            Axis.CommandRunning := FALSE;
            uiFbState := 50; (*Error state*)
            Error := TRUE;
            ErrorID := 16#06; (*Invalid input(s)*)
        END_IF;
        
    2:  IF NOT Enable THEN
            (*Send stop command*)
            usiNewCmdCount := (usiOldCmdCount + 1) MOD 16; (*MOD 16*)
            Axis.PlcToDrv.MCHeader := 16#0000; (*Reset Header*)
            Axis.PlcToDrv.MCHeader := 16#0170 + usiNewCmdCount; (*Stop command*)
            
            (*Parameter Umrechung*)
            (*Calculate parameters*)
            udiTmpDWord := REAL_TO_UDINT(Deceleration / 100); (*Deceleration*)
            Axis.PlcToDrv.MCParaWord0 := UDINT_TO_UINT(udiTmpDWord);
            Axis.PlcToDrv.MCParaWord1 := UDINT_TO_UINT(ROR(udiTmpDWord, 16));
			
			LM_UptMCI(Axis);
            
            uiFbState := 3;
        END_IF;
        
    3:  (*Prüfen ob Befehl ausgeführt ][ Check if command has been executed*)
        IF usiOldCmdCount = usiNewCmdCount AND uiCState = 16#08 AND Axis.DrvToPlc.StateVar.6 THEN
            Busy := FALSE;
            Axis.PlcToDrv.MCHeader := 16#0000 + usiNewCmdCount; (*Send no operation*)
            Axis.CommandRunning := FALSE;
            uiFbState := 0;
        END_IF;
        
    50: Error := TRUE;
        Busy := FALSE;
        Done := FALSE;
        IF NOT Enable THEN
            uiFbState := 0;
            Error := FALSE;
            ErrorID := 0;
        END_IF;
        
END_CASE;

END_FUNCTION_BLOCK

// POUs/Rotary Motors/LMmt_RotMoveInfPos
FUNCTION_BLOCK LMmt_RotMoveInfPos
VAR_INPUT
	Enable			:BOOL;	(*Enable command*)
	Velocity		:REAL;	(*[Units/s]*)
	Acceleration	:REAL;	(*[Units/s^2]*)
	Deceleration	:REAL;	(*[Units/s^2]*)
END_VAR
VAR_IN_OUT
	Axis			:tstLM_Axis; (*Axis reference*)
END_VAR
VAR_OUTPUT
	Done			:BOOL;	(*Command has been executed*)
	Busy			:BOOL;	(*Command running / FB Busy*)
	Error			:BOOL;	(*Error detected*)
	ErrorID			:UINT;	(*Error ID:
							01h: Axis not ready
 							02h: Axis already has command running
 							03h: Axis has error
 							04h: Command interrupted
 							05h: Command aborted
							06h: Invalid input(s)
							*)
END_VAR
VAR
	usiOldCmdCount 	:USINT;	(*internal -> *)
	usiNewCmdCount	:USINT;	(*internal -> *)
	uiCState		:UINT;	(*internal -> *)
	uiFbState		:UINT;	(*internal -> *)
	rTrig			:LM_R_TRIG;	(*internal -> *)
	udiTmpDWord		:UDINT;	(*internal -> *)

 	uiCmdHeader 	:UINT := 16#0CE0;	(*CommandHeader (0CExh) of the "VAI Dec=Acc VAI Inifite Motion Positive Direction (0CExh)" motion command*)
END_VAR
(*Version history:
Date         	 | Version    		| Created under     	| Author          	| Remark 
------------------------------------------------------------------------------------------------------------------------------- 
2014-oct-20   	 | 1.0.0.0     		| v3.1.4014.0			| fj  				| initial version
*)

(*Variablen ][ variables*)
usiOldCmdCount := SHR(UINT_TO_USINT(SHL(Axis.DrvToPlc.StateVar,4)),4);
uiCState := SHR(Axis.DrvToPlc.StateVar, 8);

(*Flankenerkennung am Execute Eingang*)
(*Edge detection on Execute input*)
rTrig(CLK:=Enable);
IF rTrig.Q AND uiCState = 16#08 AND NOT Axis.CommandRunning THEN (*Start command*)
	Axis.CommandRunning := TRUE;
	Busy := TRUE;
	uiFbState := 1;
ELSIF rTrig.Q AND Busy THEN (*Restart command / New rising edge on execute input*)
	Axis.CommandRunning := TRUE;
	Busy := TRUE;
	uiFbState := 1;
ELSIF rTrig.Q AND uiCState <> 16#08 THEN (*Axis not ready*)
	uiFbState := 50; (*Error state*)
	Error := TRUE;
	ErrorID := 16#01; (*Axis not ready*)
ELSIF rTrig.Q AND Axis.CommandRunning AND NOT Busy THEN (*Axis already has a command running*)
	uiFbState := 50; (*Error state*)
	Error := TRUE;
	ErrorID := 16#02; (*Axis already has a command running*)
END_IF

IF Busy AND uiCState = 16#04 THEN
	Axis.CommandRunning := FALSE;
	uiFbState := 50;
	Error := TRUE;
	ErrorID := 16#03; (*Axis has error*)
END_IF

IF Busy AND uiCState <> 16#08 THEN
	Axis.CommandRunning := FALSE;
	uiFbState := 50; (*Error state*)
	Error := TRUE;
	ErrorID := 16#04; (*Command interupted*)
ELSIF Busy AND Axis.CommandAborted THEN
	uiFbState := 50; (*Error state*)
	Error := TRUE;
	ErrorID := 16#05; (*Command aborted*)
END_IF

(*State machine*)
CASE uiFbState OF
    0:  ;
        
    1:  (*Check inputs on valid value*)
        IF (0.0 <= Velocity)
            AND (0.0 < Acceleration)
            AND (0.0 < Deceleration)
        THEN
        (*Send motion command*)
            usiNewCmdCount := (usiOldCmdCount + 1) MOD 16; (*Command counter MOD 16*)
            Axis.PlcToDrv.MCHeader := 16#0000; (*Reset Header*)
            Axis.PlcToDrv.MCHeader := uiCmdHeader + usiNewCmdCount;
            
            (*Parameter Umrechung*)
            (*Calculate parameters*)
            udiTmpDWord := REAL_TO_UDINT(Velocity / 10); (*Velocity*)
            Axis.PlcToDrv.MCParaWord0 := UDINT_TO_UINT(udiTmpDWord);
            Axis.PlcToDrv.MCParaWord1 := UDINT_TO_UINT(ROR(udiTmpDWord, 16));
            
            udiTmpDWord := REAL_TO_UDINT(Acceleration / 100); (*Acceleration*)
            Axis.PlcToDrv.MCParaWord2 := UDINT_TO_UINT(udiTmpDWord);
            Axis.PlcToDrv.MCParaWord3 := UDINT_TO_UINT(ROR(udiTmpDWord, 16));
			
			LM_UptMCI(Axis);
            
            uiFbState := 2;
        ELSE
            Axis.CommandRunning := FALSE;
            uiFbState := 50; (*Error state*)
            Error := TRUE;
            ErrorID := 16#06; (*Invalid input(s)*)
        END_IF;
        
    2:  IF NOT Enable THEN
            (*Send stop command*)
            usiNewCmdCount := (usiOldCmdCount + 1) MOD 16; (*MOD 16*)
            Axis.PlcToDrv.MCHeader := 16#0000; (*Reset Header*)
            Axis.PlcToDrv.MCHeader := 16#0170 + usiNewCmdCount; (*Stop command*)
            
            (*Parameter Umrechung*)
            (*Calculate parameters*)
            udiTmpDWord := REAL_TO_UDINT(Deceleration / 100); (*Deceleration*)
            Axis.PlcToDrv.MCParaWord0 := UDINT_TO_UINT(udiTmpDWord);
            Axis.PlcToDrv.MCParaWord1 := UDINT_TO_UINT(ROR(udiTmpDWord, 16));
			
			LM_UptMCI(Axis);
            
            uiFbState := 3;
        END_IF;
        
    3:  (*Prüfen ob Befehl ausgeführt ][ Check if command has been executed*)
        IF usiOldCmdCount = usiNewCmdCount AND uiCState = 16#08 AND Axis.DrvToPlc.StateVar.6 THEN
            Busy := FALSE;
            Axis.PlcToDrv.MCHeader := 16#0000 + usiNewCmdCount; (*Send no operation*)
            Axis.CommandRunning := FALSE;
            uiFbState := 0;
        END_IF;
        
    50: Error := TRUE;
        Busy := FALSE;
        Done := FALSE;
        IF NOT Enable THEN
            uiFbState := 0;
            Error := FALSE;
            ErrorID := 0;
        END_IF;
        
END_CASE;

END_FUNCTION_BLOCK

// POUs/Rotary Motors/LMmt_RotMoveRel
FUNCTION_BLOCK LMmt_RotMoveRel
VAR_INPUT
	Execute			:BOOL;	(*Execute command*)
	Distance		:DINT;	(*Distance in [Units]*)
	Velocity		:REAL;	(*[Units/s]*)
	Acceleration	:REAL;	(*[Units/s^2]*)
	Deceleration	:REAL;	(*[Units/s^2]*)
END_VAR
VAR_IN_OUT
	Axis			:tstLM_Axis; (*Axis reference*)
END_VAR
VAR_OUTPUT
	Done			:BOOL;	(*Command has been executed*)
	Busy			:BOOL;	(*Command running / FB Busy*)
	Error			:BOOL;	(*Error detected*)
	ErrorID			:UINT;	(*Error ID:
							01h: Axis not ready
 							02h: Axis already has command running
 							03h: Axis has error
 							04h: Command interrupted
 							05h: Command aborted
							06h: Invalid input(s)
							*)
END_VAR
VAR
	usiOldCmdCount 	:USINT;	(*internal -> *)
	usiNewCmdCount	:USINT;	(*internal -> *)
	uiCState		:UINT;	(*internal -> *)
	uiFbState		:UINT;	(*internal -> *)
	rTrig			:LM_R_TRIG;	(*internal -> *)
	udiTmpDWord		:UDINT;	(*internal -> *)

 	uiCmdHeader 	:UINT := 16#0110;	(*CommandHeader (011xh) of the "VAI Incr Dem Position (011xh)" motion command*)
END_VAR
(*Version history:
Date         	 | Version    		| Created under     	| Author          	| Remark 
------------------------------------------------------------------------------------------------------------------------------- 
2014-oct-20   	 | 1.0.0.0     		| v3.1.4014.0			| fj  				| initial version
*)

(*Variablen ][ variables*)
usiOldCmdCount := SHR(UINT_TO_USINT(SHL(Axis.DrvToPlc.StateVar,4)),4);
uiCState := SHR(Axis.DrvToPlc.StateVar, 8);

(*Flankenerkennung am Execute Eingang*)
(*Edge detection on Execute input*)
rTrig(CLK:=Execute);
IF rTrig.Q AND uiCState = 16#08 AND NOT Axis.CommandRunning THEN (*Start command*)
	Axis.CommandRunning := TRUE;
	Busy := TRUE;
	uiFbState := 1;
ELSIF rTrig.Q AND Busy THEN (*Restart command / New rising edge on execute input*)
	Axis.CommandRunning := TRUE;
	Busy := TRUE;
	uiFbState := 1;
ELSIF rTrig.Q AND uiCState <> 16#08 THEN (*Axis not ready*)
	uiFbState := 50; (*Error state*)
	Error := TRUE;
	ErrorID := 16#01; (*Axis not ready*)
ELSIF rTrig.Q AND Axis.CommandRunning AND NOT Busy THEN (*Axis already has a command running*)
	uiFbState := 50; (*Error state*)
	Error := TRUE;
	ErrorID := 16#02; (*Axis already has a command running*)
END_IF

IF Busy AND uiCState = 16#04 THEN
	Axis.CommandRunning := FALSE;
	uiFbState := 50;
	Error := TRUE;
	ErrorID := 16#03; (*Axis has error*)
END_IF

IF Busy AND uiCState <> 16#08 THEN
	Axis.CommandRunning := FALSE;
	uiFbState := 50; (*Error state*)
	Error := TRUE;
	ErrorID := 16#04; (*Command interupted*)
ELSIF Busy AND Axis.CommandAborted THEN
	uiFbState := 50; (*Error state*)
	Error := TRUE;
	ErrorID := 16#05; (*Command aborted*)
END_IF

(*State machine*)
CASE uiFbState OF
    0:  ;
        
    1:  (*Check inputs on valid value*)
        IF (-2147483648 < Distance AND Distance < 2147483647)
            AND (0.0 < Velocity)
            AND (0.0 < Acceleration)
            AND (0.0 < Deceleration)
        THEN
        (*Befehlskopf mit CMD Count berechen und senden ][ Calculate and send command header*)
            usiNewCmdCount := (usiOldCmdCount + 1) MOD 16; (*Command counter MOD 16*)
            Axis.PlcToDrv.MCHeader := 16#0000; (*Reset Header*)
            Axis.PlcToDrv.MCHeader := uiCmdHeader + usiNewCmdCount;
                      
			udiTmpDWord := DINT_TO_UDINT(Distance); (*Position increment*)
            Axis.PlcToDrv.MCParaWord0 := UDINT_TO_UINT(udiTmpDWord);
            Axis.PlcToDrv.MCParaWord1 := UDINT_TO_UINT(ROR(udiTmpDWord, 16));
            
            udiTmpDWord := DINT_TO_UDINT(REAL_TO_DINT(Velocity / 10)); (*Velocity*)
            Axis.PlcToDrv.MCParaWord2 := UDINT_TO_UINT(udiTmpDWord);
            Axis.PlcToDrv.MCParaWord3 := UDINT_TO_UINT(ROR(udiTmpDWord, 16));
            
            udiTmpDWord := DINT_TO_UDINT(REAL_TO_DINT(Acceleration / 100)); (*Acceleration*)
            Axis.PlcToDrv.MCParaWord4 := UDINT_TO_UINT(udiTmpDWord);
            Axis.PlcToDrv.MCParaWord5 := UDINT_TO_UINT(ROR(udiTmpDWord, 16));
            
            udiTmpDWord := DINT_TO_UDINT(REAL_TO_DINT(Deceleration / 100)); (*Deceleration*)
            Axis.PlcToDrv.MCParaWord6 := UDINT_TO_UINT(udiTmpDWord);
            Axis.PlcToDrv.MCParaWord7 := UDINT_TO_UINT(ROR(udiTmpDWord, 16));
			
			LM_UptMCI(Axis);
            
            uiFbState := 2;
        ELSE
            Axis.CommandRunning := FALSE;
            uiFbState := 50; (*Error state*)
            Error := TRUE;
            ErrorID := 16#06; (*Invalid input(s)*)
        END_IF;
        
    2:  (*Prüfen ob Befehl ausgeführt ][ Check if command has been executed*)
        IF usiOldCmdCount = usiNewCmdCount AND uiCState = 16#08 AND Axis.DrvToPlc.StateVar.6 THEN
            Done := TRUE;
            Busy := FALSE;
            Axis.PlcToDrv.MCHeader := 16#0000 + usiNewCmdCount; (*Send no operation*)
            Axis.CommandRunning := FALSE;
            uiFbState := 3;
        END_IF;
        
    3:  IF NOT Execute THEN
            uiFbState := 0;
            Busy := FALSE;
            Done := FALSE;
        END_IF;
        
    50: Error := TRUE;
        Busy := FALSE;
        Done := FALSE;
        IF NOT Execute THEN
            uiFbState := 0;
            Error := FALSE;
            ErrorID := 0;
        END_IF;
        
END_CASE;

END_FUNCTION_BLOCK

// POUs/Rotary Motors/LMmt_RotMoveRelJ
FUNCTION_BLOCK LMmt_RotMoveRelJ
VAR_INPUT
	Execute			:BOOL;	(*Execute command*)
	Distance		:DINT;	(*Distance in [Units]*)
	Velocity		:REAL;	(*Maximal velocity [Units/s]*)
	Acceleration	:REAL;	(*Maximal acceleration [Units/s^2]*)
	Deceleration	:REAL;	(*Maximal deceleration [Units/s^2]*)
	Jerk			:REAL;	(*Jerk [Units/s^3]*)
END_VAR
VAR_IN_OUT
	Axis			:tstLM_Axis; (*Axis reference*)
END_VAR
VAR_OUTPUT
	Done			:BOOL;	(*Command has been executed*)
	Busy			:BOOL;	(*Command running / FB Busy*)
	Error			:BOOL;	(*Error detected*)
	ErrorID			:UINT;	(*Error ID:
							01h: Axis not ready
 							02h: Axis already has command running
 							03h: Axis has error
 							04h: Command interrupted
 							05h: Command aborted
							06h: Invalid input(s)
							*)
END_VAR
VAR
	usiOldCmdCount 	:USINT;	(*internal -> *)
	usiNewCmdCount	:USINT;	(*internal -> *)
	uiCState		:UINT;	(*internal -> *)
	uiFbState		:UINT;	(*internal -> *)
	rTrig			:LM_R_TRIG;	(*internal -> *)
	udiTmpDWord		:UDINT;	(*internal -> *)

 	uiCmdHeader 	:UINT := 16#3A10; (*CommandHeader (3A1xh) of the "VAJI Increment Dem Pos (3A1xh)" motion command*)
END_VAR
(*Version history:
Date         	 | Version    		| Created under     	| Author          	| Remark 
------------------------------------------------------------------------------------------------------------------------------- 
2016-jan-05    	 | 1.0.0.0     		| v3.1.4016.12			| fj  				| initial version
*)

